C05497=1146.849,185.688,-61.263,-178.263,7.229,148.849
C05498=1146.844,185.937,-61.286,-178.260,7.230,148.849
C05499=1146.839,186.185,-61.308,-178.257,7.233,148.849
C05500=1146.835,186.434,-61.332,-178.255,7.235,148.849
C05501=1146.830,186.683,-61.355,-178.251,7.238,148.848
C05502=1146.825,186.932,-61.378,-178.249,7.240,148.848
C05503=1146.820,187.181,-61.402,-178.246,7.242,148.848
C05504=1146.816,187.430,-61.426,-178.244,7.244,148.848
C05505=1146.811,187.679,-61.449,-178.240,7.247,148.847
C05506=1146.807,187.928,-61.472,-178.238,7.249,148.847
C05507=1146.803,188.177,-61.495,-178.235,7.252,148.847
C05508=1146.798,188.426,-61.519,-178.232,7.253,148.846
C05509=1146.793,188.675,-61.542,-178.229,7.256,148.846
C05510=1146.789,188.923,-61.566,-178.227,7.258,148.846
C05511=1146.784,189.172,-61.590,-178.224,7.261,148.846
C05512=1146.780,189.421,-61.613,-178.221,7.263,148.845
C05513=1146.775,189.670,-61.636,-178.218,7.266,148.845
C05514=1146.770,189.919,-61.660,-178.216,7.267,148.845
C05515=1146.766,190.168,-61.684,-178.212,7.270,148.845
C05516=1146.761,190.417,-61.707,-178.210,7.272,148.845
C05517=1146.756,190.666,-61.730,-178.207,7.274,148.844
C05518=1146.752,190.914,-61.754,-178.205,7.277,148.844
C05519=1146.747,191.163,-61.778,-178.201,7.279,148.844
C05520=1146.743,191.412,-61.801,-178.199,7.281,148.844
C05521=1146.738,191.661,-61.825,-178.196,7.284,148.843
C05522=1146.733,191.910,-61.849,-178.194,7.286,148.843
C05523=1146.729,192.158,-61.873,-178.190,7.288,148.843
C05524=1146.724,192.407,-61.896,-178.188,7.291,148.843
C05525=1146.720,192.656,-61.919,-178.185,7.293,148.842
C05526=1146.715,192.904,-61.944,-178.182,7.296,148.842
C05527=1146.711,193.153,-61.967,-178.180,7.298,148.842
C05528=1146.706,193.402,-61.991,-178.177,7.301,148.842
C05529=1146.701,193.651,-62.014,-178.174,7.302,148.841
C05530=1146.697,193.899,-62.038,-178.171,7.305,148.841
C05531=1146.692,194.149,-62.062,-178.169,7.307,148.841
C05532=1146.688,194.398,-62.087,-178.165,7.310,148.841
C05533=1146.683,194.647,-62.110,-178.163,7.312,148.840
C05534=1146.679,194.895,-62.134,-178.160,7.314,148.840
C05535=1146.674,195.144,-62.158,-178.157,7.317,148.840
C05536=1146.670,195.393,-62.182,-178.154,7.319,148.840
C05537=1146.665,195.642,-62.205,-178.151,7.322,148.840
C05538=1146.661,195.890,-62.229,-178.149,7.324,148.839
C05539=1146.655,196.139,-62.253,-178.146,7.326,148.839
C05540=1146.651,196.388,-62.277,-178.143,7.328,148.839
C05541=1146.647,196.637,-62.302,-178.140,7.331,148.839
C05542=1146.642,196.886,-62.325,-178.138,7.333,148.838
C05543=1146.638,197.134,-62.349,-178.135,7.336,148.838
C05544=1146.632,197.384,-62.373,-178.132,7.338,148.838
C05545=1146.628,197.632,-62.397,-178.129,7.340,148.838
C05546=1146.624,197.881,-62.421,-178.127,7.343,148.838
C05547=1146.620,198.130,-62.445,-178.124,7.345,148.837
C05548=1146.615,198.379,-62.469,-178.121,7.348,148.837
C05549=1146.610,198.627,-62.494,-178.118,7.351,148.837
C05550=1146.606,198.876,-62.518,-178.116,7.353,148.837
C05551=1146.601,199.125,-62.541,-178.112,7.355,148.836
C05552=1146.596,199.374,-62.566,-178.110,7.357,148.836
C05553=1146.592,199.623,-62.590,-178.107,7.360,148.836
C05554=1146.588,199.871,-62.614,-178.104,7.363,148.836
C05555=1146.583,200.120,-62.638,-178.101,7.364,148.835
C05556=1146.578,200.369,-62.662,-178.099,7.367,148.835
C05557=1146.574,200.618,-62.687,-178.096,7.369,148.835
C05558=1146.570,200.866,-62.711,-178.093,7.372,148.835
C05559=1146.564,201.115,-62.735,-178.090,7.375,148.834
C05560=1146.560,201.364,-62.759,-178.088,7.377,148.834
C05561=1146.555,201.613,-62.783,-178.085,7.380,148.834
C05562=1146.551,201.862,-62.808,-178.082,7.381,148.834
C05563=1146.546,202.110,-62.832,-178.079,7.384,148.834
C05564=1146.542,202.359,-62.856,-178.076,7.387,148.833
C05565=1146.537,202.608,-62.881,-178.074,7.389,148.833
C05566=1146.533,202.857,-62.905,-178.071,7.391,148.833
C05567=1146.528,203.105,-62.930,-178.068,7.394,148.833
C05568=1146.524,203.354,-62.954,-178.066,7.397,148.833
C05569=1146.520,203.603,-62.978,-178.062,7.399,148.832
C05570=1146.515,203.852,-63.003,-178.060,7.401,148.832
C05571=1146.510,204.100,-63.027,-178.057,7.404,148.832
C05572=1146.506,204.350,-63.052,-178.054,7.407,148.832
C05573=1146.501,204.598,-63.076,-178.051,7.408,148.832
C05574=1146.496,204.847,-63.101,-178.049,7.411,148.831
C05575=1146.492,205.095,-63.125,-178.046,7.413,148.831
C05576=1146.488,205.344,-63.149,-178.043,7.416,148.831
C05577=1146.483,205.593,-63.174,-178.040,7.419,148.831
C05578=1146.478,205.841,-63.198,-178.038,7.421,148.831
C05579=1146.474,206.091,-63.223,-178.035,7.424,148.830
C05580=1146.469,206.339,-63.248,-178.032,7.426,148.830
C05581=1146.464,206.588,-63.272,-178.029,7.428,148.830
C05582=1146.460,206.837,-63.297,-178.027,7.431,148.830
C05583=1146.455,207.086,-63.321,-178.023,7.434,148.830
C05584=1146.451,207.334,-63.346,-178.021,7.436,148.829
C05585=1146.447,207.583,-63.371,-178.018,7.439,148.829
C05586=1146.442,207.832,-63.395,-178.015,7.441,148.829
C05587=1146.438,208.081,-63.420,-178.013,7.443,148.829
C05588=1146.433,208.330,-63.445,-178.010,7.446,148.829
C05589=1146.428,208.578,-63.469,-178.007,7.449,148.828
C05590=1146.424,208.827,-63.494,-178.004,7.451,148.828
C05591=1146.419,209.075,-63.519,-178.001,7.453,148.828
C05592=1146.415,209.346,-63.546,-177.998,7.456,148.828
C05593=1146.409,209.616,-63.573,-177.995,7.459,148.828
C05594=1146.405,209.887,-63.600,-177.992,7.462,148.827
C05595=1146.400,210.158,-63.627,-177.989,7.464,148.827
C05596=1146.395,210.407,-63.652,-177.986,7.467,148.827
C05597=1146.391,210.655,-63.676,-177.984,7.469,148.827
C05598=1146.387,210.904,-63.701,-177.981,7.472,148.827
C05599=1146.381,211.153,-63.726,-177.978,7.475,148.827
C05600=1146.377,211.401,-63.752,-177.976,7.477,148.826
C05601=1146.373,211.650,-63.776,-177.973,7.480,148.826
C05602=1146.368,211.899,-63.801,-177.970,7.483,148.826
C05603=1146.363,212.148,-63.826,-177.968,7.485,148.826
C05604=1146.359,212.396,-63.850,-177.964,7.487,148.826
C05605=1146.355,212.645,-63.876,-177.961,7.490,148.825
C05606=1146.350,212.894,-63.901,-177.959,7.492,148.825
C05607=1146.346,213.143,-63.925,-177.956,7.495,148.825
C05608=1146.341,213.391,-63.951,-177.953,7.498,148.825
C05609=1146.336,213.640,-63.976,-177.950,7.501,148.825
C05610=1146.332,213.888,-64.001,-177.948,7.502,148.824
C05611=1146.327,214.138,-64.026,-177.945,7.505,148.824
C05612=1146.323,214.386,-64.051,-177.942,7.508,148.824
C05613=1146.319,214.635,-64.076,-177.939,7.510,148.824
C05614=1146.314,214.883,-64.101,-177.937,7.513,148.824
C05615=1146.309,215.132,-64.127,-177.934,7.516,148.824
C05616=1146.304,215.381,-64.152,-177.931,7.519,148.824
C05617=1146.301,215.629,-64.177,-177.928,7.520,148.823
C05618=1146.296,215.878,-64.202,-177.926,7.523,148.823
C05619=1146.291,216.127,-64.227,-177.923,7.526,148.823
C05620=1146.287,216.376,-64.252,-177.920,7.528,148.823
C05621=1146.282,216.624,-64.278,-177.917,7.531,148.823
C05622=1146.278,216.873,-64.304,-177.914,7.534,148.823
C05623=1146.274,217.121,-64.328,-177.911,7.536,148.822
C05624=1146.269,217.370,-64.353,-177.909,7.539,148.822
C05625=1146.264,217.618,-64.379,-177.906,7.541,148.822
C05626=1146.260,217.868,-64.404,-177.903,7.544,148.822
C05627=1146.256,218.117,-64.430,-177.900,7.547,148.822
C05628=1146.251,218.365,-64.455,-177.898,7.549,148.822
C05629=1146.247,218.613,-64.481,-177.895,7.552,148.821
C05630=1146.242,218.863,-64.506,-177.892,7.554,148.821
C05631=1146.237,219.111,-64.531,-177.889,7.557,148.821
C05632=1146.233,219.360,-64.557,-177.887,7.560,148.821
C05633=1146.228,219.608,-64.582,-177.884,7.562,148.821
C05634=1146.224,219.857,-64.607,-177.881,7.565,148.820
C05635=1146.220,220.106,-64.632,-177.878,7.568,148.820
C05636=1146.215,220.354,-64.658,-177.876,7.570,148.820
C05637=1146.211,220.603,-64.684,-177.873,7.573,148.820
C05638=1146.207,220.851,-64.709,-177.870,7.576,148.820
C05639=1146.202,221.100,-64.735,-177.867,7.578,148.820
C05640=1146.198,221.348,-64.760,-177.865,7.581,148.820
C05641=1146.193,221.598,-64.786,-177.862,7.583,148.820
C05642=1146.188,221.846,-64.811,-177.859,7.586,148.819
C05643=1146.184,222.095,-64.837,-177.856,7.589,148.819
C05644=1146.179,222.344,-64.863,-177.854,7.591,148.819
C05645=1146.175,222.592,-64.888,-177.851,7.594,148.819
C05646=1146.170,222.841,-64.914,-177.848,7.597,148.819
C05647=1146.166,223.090,-64.940,-177.845,7.599,148.819
C05648=1146.161,223.338,-64.965,-177.842,7.602,148.818
C05649=1146.157,223.586,-64.991,-177.840,7.604,148.818
C05650=1146.153,223.835,-65.017,-177.837,7.607,148.818
C05651=1146.149,224.084,-65.043,-177.834,7.610,148.818
C05652=1146.144,224.332,-65.068,-177.831,7.613,148.818
C05653=1146.139,224.581,-65.094,-177.828,7.616,148.818
C05654=1146.135,224.830,-65.120,-177.826,7.618,148.818
C05655=1146.130,225.079,-65.146,-177.823,7.620,148.817
C05656=1146.126,225.327,-65.171,-177.820,7.623,148.817
C05657=1146.121,225.576,-65.197,-177.817,7.626,148.817
C05658=1146.117,225.824,-65.223,-177.814,7.629,148.817
C05659=1146.112,226.073,-65.250,-177.812,7.631,148.817
C05660=1146.108,226.321,-65.275,-177.809,7.634,148.817
C05661=1146.103,226.570,-65.301,-177.806,7.637,148.817
C05662=1146.099,226.819,-65.327,-177.803,7.640,148.816
C05663=1146.095,227.068,-65.352,-177.800,7.643,148.816
C05664=1146.089,227.316,-65.378,-177.798,7.645,148.816
C05665=1146.085,227.564,-65.405,-177.795,7.647,148.816
C05666=1146.081,227.813,-65.431,-177.792,7.650,148.816
C05667=1146.077,228.062,-65.456,-177.789,7.653,148.816
C05668=1146.072,228.311,-65.483,-177.787,7.656,148.816
C05669=1146.068,228.558,-65.509,-177.784,7.658,148.816
C05670=1146.063,228.807,-65.534,-177.782,7.661,148.816
C05671=1146.059,229.056,-65.560,-177.778,7.664,148.815
C05672=1146.054,229.305,-65.587,-177.776,7.667,148.815
C05673=1146.050,229.553,-65.613,-177.773,7.670,148.815
C05674=1146.046,229.802,-65.639,-177.770,7.672,148.815
C05675=1146.041,230.051,-65.665,-177.768,7.675,148.815
C05676=1146.036,230.299,-65.691,-177.765,7.677,148.815
C05677=1146.032,230.548,-65.717,-177.762,7.680,148.814
C05678=1146.027,230.797,-65.743,-177.759,7.683,148.814
C05679=1146.023,231.045,-65.770,-177.756,7.686,148.814
C05680=1146.019,231.294,-65.796,-177.753,7.689,148.814
C05681=1146.014,231.542,-65.823,-177.751,7.691,148.814
C05682=1146.010,231.791,-65.848,-177.748,7.694,148.814
C05683=1146.006,232.039,-65.875,-177.745,7.696,148.814
C05684=1146.001,232.288,-65.901,-177.742,7.699,148.814
C05685=1145.997,232.536,-65.927,-177.739,7.702,148.814
C05686=1145.992,232.785,-65.954,-177.737,7.705,148.813
C05687=1145.988,233.034,-65.979,-177.734,7.708,148.813
C05688=1145.983,233.282,-66.006,-177.732,7.710,148.813
C05689=1145.979,233.531,-66.032,-177.729,7.713,148.813
C05690=1145.975,233.779,-66.059,-177.726,7.716,148.813
C05691=1145.970,234.028,-66.086,-177.723,7.719,148.813
C05692=1145.966,234.276,-66.111,-177.720,7.722,148.813
C05693=1145.961,234.525,-66.139,-177.717,7.724,148.813
C05694=1145.957,234.774,-66.164,-177.714,7.727,148.813
C05695=1145.952,235.022,-66.191,-177.712,7.729,148.812
C05696=1145.948,235.294,-66.220,-177.709,7.733,148.812
C05697=1145.943,235.566,-66.249,-177.706,7.736,148.812
C05698=1145.938,235.837,-66.278,-177.703,7.739,148.812
C05699=1145.934,236.109,-66.307,-177.700,7.742,148.812
C05700=1145.929,236.358,-66.334,-177.697,7.745,148.812
C05701=1145.924,236.607,-66.361,-177.694,7.747,148.812
C05702=1145.920,236.855,-66.387,-177.692,7.750,148.812
C05703=1145.915,237.104,-66.413,-177.689,7.753,148.812
C05704=1145.911,237.352,-66.440,-177.686,7.756,148.811
C05705=1145.907,237.601,-66.467,-177.683,7.759,148.811
C05706=1145.903,237.849,-66.493,-177.680,7.762,148.811
C05707=1145.898,238.098,-66.520,-177.678,7.764,148.811
C05708=1145.893,238.347,-66.547,-177.675,7.767,148.811
C05709=1145.889,238.595,-66.573,-177.672,7.770,148.811
C05710=1145.885,238.843,-66.600,-177.669,7.773,148.811
C05711=1145.880,239.093,-66.627,-177.667,7.776,148.811
C05712=1145.876,239.341,-66.653,-177.664,7.778,148.811
C05713=1145.871,239.589,-66.680,-177.661,7.781,148.811
C05714=1145.866,239.838,-66.707,-177.658,7.784,148.810
C05715=1145.862,240.086,-66.734,-177.656,7.787,148.810
C05716=1145.858,240.334,-66.761,-177.653,7.790,148.810
C05717=1145.853,240.583,-66.788,-177.650,7.792,148.810
C05718=1145.849,240.831,-66.814,-177.647,7.795,148.810
C05719=1145.844,241.080,-66.841,-177.644,7.798,148.810
C05720=1145.840,241.329,-66.868,-177.642,7.801,148.810
C05721=1145.836,241.577,-66.894,-177.639,7.804,148.810
C05722=1145.832,241.826,-66.922,-177.636,7.807,148.810
C05723=1145.827,242.075,-66.949,-177.633,7.809,148.810
C05724=1145.822,242.323,-66.976,-177.631,7.812,148.809
C05725=1145.818,242.571,-67.002,-177.628,7.815,148.809
C05726=1145.814,242.820,-67.029,-177.625,7.818,148.809
C05727=1145.809,243.068,-67.056,-177.622,7.821,148.809
C05728=1145.804,243.317,-67.083,-177.619,7.824,148.809
C05729=1145.800,243.565,-67.110,-177.617,7.826,148.809
C05730=1145.797,243.813,-67.138,-177.614,7.829,148.809
C05731=1145.792,244.062,-67.165,-177.612,7.832,148.809
C05732=1145.787,244.310,-67.192,-177.609,7.835,148.809
C05733=1145.783,244.559,-67.219,-177.606,7.838,148.809
C05734=1145.778,244.807,-67.246,-177.603,7.841,148.809
C05735=1145.774,245.056,-67.273,-177.600,7.844,148.809
C05736=1145.770,245.305,-67.300,-177.598,7.847,148.809
C05737=1145.765,245.553,-67.327,-177.595,7.850,148.808
C05738=1145.761,245.801,-67.355,-177.592,7.853,148.808
C05739=1145.756,246.050,-67.382,-177.589,7.855,148.808
C05740=1145.752,246.298,-67.409,-177.586,7.858,148.808
C05741=1145.748,246.547,-67.437,-177.584,7.861,148.808
C05742=1145.743,246.796,-67.464,-177.581,7.864,148.808
C05743=1145.739,247.044,-67.491,-177.578,7.867,148.808
C05744=1145.735,247.292,-67.518,-177.575,7.870,148.808
C05745=1145.731,247.541,-67.545,-177.573,7.873,148.808
C05746=1145.726,247.790,-67.572,-177.570,7.875,148.808
C05747=1145.722,248.038,-67.600,-177.568,7.878,148.808
C05748=1145.717,248.286,-67.627,-177.565,7.881,148.808
C05749=1145.713,248.535,-67.655,-177.562,7.884,148.808
C05750=1145.709,248.783,-67.682,-177.559,7.887,148.807
C05751=1145.704,249.032,-67.709,-177.556,7.890,148.807
C05752=1145.699,249.280,-67.736,-177.554,7.893,148.807
C05753=1145.696,249.529,-67.765,-177.551,7.896,148.807
C05754=1145.691,249.777,-67.792,-177.548,7.898,148.807
C05755=1145.687,250.025,-67.819,-177.545,7.901,148.807
C05756=1145.682,250.274,-67.847,-177.542,7.904,148.807
C05757=1145.678,250.522,-67.875,-177.540,7.907,148.807
C05758=1145.674,250.771,-67.902,-177.537,7.910,148.807
C05759=1145.669,251.019,-67.929,-177.534,7.913,148.807
C05760=1145.665,251.268,-67.957,-177.531,7.916,148.807
C05761=1145.660,251.516,-67.985,-177.529,7.919,148.807
C05762=1145.655,251.764,-68.012,-177.526,7.922,148.807
C05763=1145.651,252.014,-68.040,-177.523,7.925,148.807
C05764=1145.647,252.261,-68.068,-177.520,7.928,148.806
C05765=1145.643,252.509,-68.095,-177.517,7.931,148.806
C05766=1145.639,252.758,-68.123,-177.515,7.934,148.806
C05767=1145.634,253.006,-68.151,-177.512,7.937,148.806
C05768=1145.630,253.255,-68.178,-177.509,7.939,148.806
C05769=1145.626,253.503,-68.206,-177.506,7.942,148.806
C05770=1145.620,253.752,-68.233,-177.503,7.945,148.806
C05771=1145.616,254.000,-68.261,-177.501,7.949,148.806
C05772=1145.612,254.249,-68.289,-177.498,7.951,148.806
C05773=1145.608,254.497,-68.316,-177.496,7.954,148.806
C05774=1145.604,254.746,-68.345,-177.493,7.957,148.806
C05775=1145.600,254.994,-68.372,-177.490,7.960,148.806
C05776=1145.594,255.242,-68.400,-177.487,7.963,148.806
C05777=1145.590,255.491,-68.428,-177.484,7.966,148.806
C05778=1145.586,255.739,-68.456,-177.482,7.969,148.806
C05779=1145.582,255.987,-68.484,-177.479,7.972,148.806
C05780=1145.577,256.236,-68.512,-177.476,7.975,148.806
C05781=1145.573,256.484,-68.539,-177.473,7.978,148.806
C05782=1145.569,256.733,-68.568,-177.470,7.981,148.805
C05783=1145.564,256.981,-68.595,-177.468,7.984,148.806
C05784=1145.560,257.230,-68.623,-177.465,7.987,148.806
C05785=1145.555,257.478,-68.651,-177.463,7.990,148.805
C05786=1145.552,257.727,-68.679,-177.460,7.993,148.805
C05787=1145.547,257.975,-68.708,-177.457,7.996,148.805
C05788=1145.543,258.223,-68.736,-177.454,7.999,148.805
C05789=1145.538,258.471,-68.764,-177.451,8.002,148.805
C05790=1145.534,258.720,-68.792,-177.449,8.005,148.805
C05791=1145.529,258.969,-68.819,-177.446,8.007,148.805
C05792=1145.526,259.217,-68.848,-177.444,8.011,148.805
C05793=1145.520,259.465,-68.876,-177.441,8.014,148.805
C05794=1145.517,259.714,-68.904,-177.438,8.017,148.805
C05795=1145.512,259.962,-68.932,-177.435,8.020,148.805
C05796=1145.508,260.211,-68.961,-177.432,8.022,148.805
C05797=1145.503,260.459,-68.988,-177.430,8.025,148.805
C05798=1145.500,260.707,-69.017,-177.427,8.028,148.805
C05799=1145.495,260.955,-69.045,-177.423,8.032,148.805
C05800=1145.490,261.229,-69.076,-177.421,8.035,148.805
C05801=1145.485,261.502,-69.107,-177.418,8.038,148.805
C05802=1145.481,261.776,-69.139,-177.415,8.042,148.805
C05803=1145.476,262.049,-69.169,-177.412,8.045,148.805
C05804=1145.471,262.297,-69.198,-177.409,8.048,148.805
C05805=1145.467,262.546,-69.226,-177.407,8.051,148.805
C05806=1145.463,262.795,-69.255,-177.404,8.054,148.805
C05807=1145.458,263.043,-69.282,-177.400,8.057,148.805
C05808=1145.454,263.291,-69.311,-177.398,8.061,148.805
C05809=1145.450,263.539,-69.340,-177.395,8.064,148.805
C05810=1145.445,263.788,-69.368,-177.393,8.067,148.805
C05811=1145.441,264.035,-69.396,-177.390,8.069,148.805
C05812=1145.437,264.284,-69.425,-177.387,8.072,148.805
C05813=1145.433,264.533,-69.453,-177.384,8.075,148.804
C05814=1145.428,264.781,-69.482,-177.382,8.079,148.805
C05815=1145.424,265.029,-69.511,-177.379,8.082,148.805
C05816=1145.419,265.277,-69.539,-177.376,8.084,148.805
C05817=1145.415,265.526,-69.567,-177.374,8.087,148.804
C05818=1145.411,265.774,-69.596,-177.371,8.090,148.804
C05819=1145.406,266.022,-69.625,-177.368,8.094,148.805
C05820=1145.402,266.271,-69.653,-177.366,8.097,148.804
C05821=1145.398,266.520,-69.681,-177.363,8.099,148.804
C05822=1145.393,266.767,-69.710,-177.359,8.103,148.804
C05823=1145.389,267.016,-69.739,-177.357,8.106,148.804
C05824=1145.385,267.264,-69.768,-177.354,8.109,148.805
C05825=1145.380,267.512,-69.796,-177.352,8.112,148.804
C05826=1145.376,267.761,-69.825,-177.349,8.115,148.804
C05827=1145.372,268.009,-69.854,-177.346,8.118,148.804
C05828=1145.367,268.257,-69.882,-177.344,8.121,148.804
C05829=1145.363,268.506,-69.911,-177.341,8.124,148.804
C05830=1145.359,268.754,-69.940,-177.338,8.127,148.804
C05831=1145.354,269.002,-69.968,-177.335,8.130,148.804
C05832=1145.351,269.250,-69.997,-177.333,8.133,148.804
C05833=1145.346,269.499,-70.026,-177.330,8.137,148.804
C05834=1145.341,269.747,-70.055,-177.327,8.140,148.804
C05835=1145.337,269.996,-70.084,-177.324,8.143,148.804
C05836=1145.334,270.244,-70.113,-177.321,8.146,148.804
C05837=1145.329,270.493,-70.141,-177.319,8.149,148.804
C05838=1145.324,270.740,-70.170,-177.316,8.152,148.804
C05839=1145.320,270.989,-70.199,-177.313,8.155,148.804
C05840=1145.316,271.237,-70.228,-177.311,8.158,148.804
C05841=1145.312,271.485,-70.258,-177.308,8.161,148.804
C05842=1145.307,271.733,-70.286,-177.305,8.164,148.804
C05843=1145.303,271.982,-70.315,-177.302,8.168,148.804
C05844=1145.299,272.230,-70.345,-177.300,8.171,148.805
C05845=1145.295,272.479,-70.373,-177.297,8.174,148.804
C05846=1145.290,272.726,-70.402,-177.294,8.177,148.804
C05847=1145.286,272.974,-70.432,-177.291,8.180,148.804
C05848=1145.281,273.223,-70.460,-177.289,8.183,148.805
C05849=1145.277,273.472,-70.490,-177.286,8.186,148.804
C05850=1145.273,273.720,-70.519,-177.284,8.189,148.804
C05851=1145.268,273.968,-70.548,-177.281,8.193,148.805
C05852=1145.265,274.216,-70.576,-177.278,8.196,148.805
C05853=1145.260,274.464,-70.606,-177.275,8.199,148.805
C05854=1145.256,274.712,-70.635,-177.272,8.202,148.804
C05855=1145.252,274.961,-70.664,-177.270,8.205,148.805
C05856=1145.248,275.210,-70.693,-177.267,8.208,148.805
C05857=1145.243,275.457,-70.723,-177.264,8.211,148.805
C05858=1145.239,275.705,-70.752,-177.262,8.215,148.805
C05859=1145.234,275.954,-70.781,-177.259,8.218,148.805
C05860=1145.230,276.202,-70.811,-177.256,8.221,148.805
C05861=1145.226,276.451,-70.840,-177.254,8.224,148.805
C05862=1145.222,276.699,-70.869,-177.251,8.227,148.805
C05863=1145.217,276.947,-70.899,-177.248,8.230,148.805
C05864=1145.213,277.196,-70.928,-177.246,8.234,148.805
C05865=1145.208,277.443,-70.957,-177.243,8.237,148.805
C05866=1145.204,277.692,-70.987,-177.240,8.240,148.805
C05867=1145.200,277.940,-71.016,-177.237,8.244,148.805
C05868=1145.196,278.188,-71.045,-177.234,8.246,148.805
C05869=1145.192,278.436,-71.075,-177.232,8.249,148.805
C05870=1145.187,278.685,-71.104,-177.229,8.253,148.805
C05871=1145.183,278.933,-71.134,-177.227,8.256,148.805
C05872=1145.179,279.181,-71.163,-177.223,8.259,148.805
C05873=1145.175,279.429,-71.193,-177.221,8.263,148.805
C05874=1145.171,279.678,-71.222,-177.218,8.266,148.805
C05875=1145.167,279.926,-71.252,-177.215,8.268,148.805
C05876=1145.162,280.174,-71.281,-177.213,8.272,148.805
C05877=1145.158,280.422,-71.311,-177.210,8.275,148.805
C05878=1145.154,280.671,-71.340,-177.207,8.279,148.805
C05879=1145.149,280.919,-71.370,-177.204,8.282,148.805
C05880=1145.145,281.166,-71.400,-177.202,8.285,148.805
C05881=1145.140,281.415,-71.429,-177.199,8.288,148.805
C05882=1145.136,281.663,-71.459,-177.197,8.291,148.805
C05883=1145.132,281.911,-71.488,-177.194,8.294,148.805
C05884=1145.128,282.159,-71.518,-177.191,8.298,148.805
C05885=1145.124,282.408,-71.547,-177.188,8.301,148.805
C05886=1145.119,282.656,-71.578,-177.186,8.304,148.806
C05887=1145.115,282.904,-71.607,-177.183,8.307,148.806
C05888=1145.111,283.152,-71.637,-177.181,8.310,148.806
C05889=1145.107,283.400,-71.666,-177.178,8.313,148.806
C05890=1145.102,283.648,-71.697,-177.175,8.317,148.806
C05891=1145.098,283.897,-71.726,-177.172,8.320,148.806
C05892=1145.094,284.145,-71.756,-177.169,8.323,148.806
C05893=1145.090,284.393,-71.786,-177.167,8.326,148.806
C05894=1145.085,284.642,-71.817,-177.164,8.329,148.806
C05895=1145.081,284.890,-71.846,-177.161,8.333,148.806
C05896=1145.077,285.138,-71.876,-177.159,8.336,148.806
C05897=1145.073,285.386,-71.906,-177.156,8.339,148.806
C05898=1145.068,285.635,-71.936,-177.154,8.343,148.806
C05899=1145.064,285.882,-71.966,-177.151,8.345,148.806
C05900=1145.060,286.130,-71.995,-177.148,8.350,148.806
C05901=1145.056,286.378,-72.026,-177.145,8.352,148.806
C05902=1145.051,286.627,-72.055,-177.143,8.356,148.806
C05903=1145.048,286.874,-72.086,-177.140,8.359,148.806
C05904=1145.042,287.151,-72.119,-177.137,8.363,148.807
C05905=1145.038,287.426,-72.153,-177.134,8.367,148.807
C05906=1145.033,287.702,-72.185,-177.131,8.369,148.807
C05907=1145.029,287.976,-72.219,-177.128,8.374,148.807
C05908=1145.024,288.225,-72.249,-177.125,8.376,148.807
C05909=1145.020,288.473,-72.279,-177.123,8.380,148.807
C05910=1145.015,288.721,-72.310,-177.120,8.383,148.807
C05911=1145.012,288.970,-72.340,-177.117,8.387,148.807
C05912=1145.008,289.217,-72.370,-177.114,8.390,148.807
C05913=1145.003,289.466,-72.400,-177.112,8.393,148.807
C05914=1144.999,289.713,-72.430,-177.109,8.397,148.807
C05915=1144.995,289.961,-72.461,-177.106,8.400,148.807
C05916=1144.990,290.210,-72.490,-177.104,8.403,148.807
C05917=1144.986,290.458,-72.521,-177.101,8.406,148.807
C05918=1144.982,290.706,-72.552,-177.098,8.409,148.807
C05919=1144.978,290.955,-72.582,-177.096,8.413,148.808
C05920=1144.974,291.202,-72.612,-177.093,8.416,148.808
C05921=1144.969,291.450,-72.642,-177.090,8.419,148.808
C05922=1144.965,291.698,-72.672,-177.088,8.422,148.808
C05923=1144.961,291.947,-72.703,-177.085,8.426,148.808
C05924=1144.957,292.195,-72.733,-177.082,8.429,148.808
C05925=1144.952,292.443,-72.764,-177.080,8.433,148.808
C05926=1144.949,292.690,-72.794,-177.077,8.436,148.808
C05927=1144.944,292.940,-72.825,-177.074,8.440,148.808
C05928=1144.940,293.187,-72.855,-177.072,8.443,148.808
C05929=1144.936,293.435,-72.886,-177.069,8.446,148.808
C05930=1144.931,293.683,-72.916,-177.067,8.449,148.809
C05931=1144.928,293.931,-72.947,-177.063,8.453,148.809
C05932=1144.923,294.179,-72.978,-177.061,8.456,148.809
C05933=1144.919,294.428,-73.007,-177.058,8.459,148.809
C05934=1144.914,294.676,-73.038,-177.056,8.462,148.809
C05935=1144.910,294.924,-73.069,-177.053,8.466,148.809
C05936=1144.907,295.172,-73.099,-177.050,8.469,148.809
C05937=1144.902,295.420,-73.130,-177.048,8.473,148.809
C05938=1144.898,295.669,-73.161,-177.045,8.476,148.809
C05939=1144.894,295.916,-73.191,-177.042,8.480,148.809
C05940=1144.889,296.164,-73.222,-177.039,8.483,148.809
C05941=1144.886,296.412,-73.252,-177.037,8.486,148.810
C05942=1144.882,296.661,-73.283,-177.035,8.489,148.810
C05943=1144.877,296.908,-73.314,-177.031,8.493,148.810
C05944=1144.872,297.156,-73.345,-177.029,8.496,148.810
C05945=1144.869,297.405,-73.375,-177.026,8.499,148.810
C05946=1144.864,297.653,-73.406,-177.023,8.503,148.810
C05947=1144.860,297.901,-73.437,-177.021,8.506,148.810
C05948=1144.856,298.149,-73.468,-177.018,8.509,148.810
C05949=1144.852,298.396,-73.499,-177.016,8.513,148.810
C05950=1144.848,298.644,-73.530,-177.013,8.517,148.811
C05951=1144.844,298.893,-73.561,-177.010,8.520,148.811
C05952=1144.839,299.141,-73.591,-177.008,8.523,148.811
C05953=1144.836,299.389,-73.622,-177.004,8.527,148.811
C05954=1144.831,299.637,-73.653,-177.002,8.530,148.811
C05955=1144.827,299.885,-73.684,-177.000,8.533,148.811
C05956=1144.823,300.133,-73.715,-176.997,8.536,148.811
C05957=1144.818,300.381,-73.746,-176.994,8.540,148.811
C05958=1144.814,300.630,-73.777,-176.992,8.543,148.811
C05959=1144.810,300.878,-73.807,-176.989,8.546,148.811
C05960=1144.806,301.125,-73.839,-176.986,8.550,148.812
C05961=1144.802,301.374,-73.870,-176.984,8.554,148.812
C05962=1144.797,301.621,-73.901,-176.981,8.557,148.812
C05963=1144.794,301.870,-73.933,-176.978,8.561,148.812
C05964=1144.789,302.117,-73.963,-176.976,8.564,148.812
C05965=1144.784,302.365,-73.994,-176.973,8.567,148.812
C05966=1144.781,302.613,-74.026,-176.971,8.570,148.812
C05967=1144.776,302.861,-74.057,-176.968,8.574,148.812
C05968=1144.772,303.110,-74.088,-176.965,8.577,148.812
C05969=1144.768,303.357,-74.119,-176.963,8.580,148.813
C05970=1144.764,303.606,-74.150,-176.960,8.585,148.813
C05971=1144.760,303.853,-74.181,-176.957,8.588,148.813
C05972=1144.756,304.102,-74.213,-176.955,8.591,148.813
C05973=1144.752,304.350,-74.243,-176.952,8.595,148.813
C05974=1144.748,304.598,-74.275,-176.949,8.598,148.813
C05975=1144.743,304.846,-74.306,-176.947,8.601,148.813
C05976=1144.739,305.093,-74.337,-176.944,8.605,148.814
C05977=1144.735,305.342,-74.369,-176.941,8.608,148.814
C05978=1144.731,305.589,-74.400,-176.939,8.612,148.814
C05979=1144.726,305.838,-74.432,-176.936,8.615,148.814
C05980=1144.722,306.086,-74.464,-176.933,8.619,148.814
C05981=1144.718,306.333,-74.495,-176.931,8.622,148.814
C05982=1144.714,306.582,-74.526,-176.928,8.626,148.815
C05983=1144.710,306.829,-74.558,-176.925,8.629,148.815
C05984=1144.706,307.078,-74.589,-176.923,8.632,148.815
C05985=1144.701,307.325,-74.620,-176.920,8.636,148.815
C05986=1144.698,307.573,-74.652,-176.918,8.640,148.815
C05987=1144.693,307.821,-74.683,-176.915,8.643,148.815
C05988=1144.689,308.069,-74.715,-176.912,8.647,148.815
C05989=1144.685,308.317,-74.746,-176.910,8.650,148.815
C05990=1144.680,308.566,-74.778,-176.907,8.653,148.816
C05991=1144.676,308.814,-74.810,-176.904,8.657,148.816
C05992=1144.672,309.061,-74.841,-176.902,8.660,148.816
C05993=1144.668,309.309,-74.873,-176.899,8.663,148.816
C05994=1144.664,309.557,-74.904,-176.896,8.667,148.816
C05995=1144.660,309.805,-74.936,-176.894,8.671,148.816
C05996=1144.656,310.053,-74.968,-176.891,8.675,148.816
C05997=1144.651,310.301,-75.000,-176.888,8.678,148.817
C05998=1144.647,310.549,-75.031,-176.886,8.681,148.817
C05999=1144.643,310.797,-75.062,-176.883,8.685,148.817
C06000=1144.639,311.045,-75.094,-176.881,8.688,148.817
C06001=1144.635,311.293,-75.127,-176.878,8.692,148.817
C06002=1144.631,311.541,-75.158,-176.875,8.695,148.817
C06003=1144.627,311.789,-75.190,-176.873,8.699,148.818
C06004=1144.623,312.037,-75.222,-176.870,8.702,148.818
C06005=1144.618,312.284,-75.254,-176.867,8.706,148.818
C06006=1144.614,312.533,-75.285,-176.865,8.709,148.818
C06007=1144.610,312.781,-75.317,-176.862,8.713,148.818
C06008=1144.606,313.059,-75.352,-176.859,8.717,148.818
C06009=1144.601,313.336,-75.389,-176.857,8.720,148.819
C06010=1144.597,313.614,-75.424,-176.854,8.724,148.819
C06011=1144.592,313.892,-75.460,-176.851,8.729,148.819
C06012=1144.587,314.139,-75.492,-176.848,8.733,148.819
C06013=1144.584,314.387,-75.524,-176.845,8.736,148.819
C06014=1144.579,314.635,-75.556,-176.843,8.739,148.820
C06015=1144.575,314.883,-75.588,-176.840,8.743,148.820
C06016=1144.571,315.131,-75.619,-176.837,8.746,148.820
C06017=1144.567,315.379,-75.652,-176.835,8.750,148.820
C06018=1144.563,315.627,-75.684,-176.832,8.754,148.820
C06019=1144.559,315.875,-75.715,-176.830,8.757,148.820
C06020=1144.555,316.122,-75.748,-176.827,8.761,148.821
C06021=1144.551,316.370,-75.780,-176.825,8.764,148.821
C06022=1144.546,316.619,-75.813,-176.822,8.768,148.821
C06023=1144.542,316.866,-75.844,-176.819,8.771,148.821
C06024=1144.538,317.114,-75.877,-176.817,8.774,148.821
C06025=1144.534,317.362,-75.908,-176.814,8.779,148.821
C06026=1144.531,317.610,-75.941,-176.811,8.782,148.822
C06027=1144.526,317.858,-75.973,-176.808,8.786,148.822
C06028=1144.522,318.105,-76.005,-176.806,8.789,148.822
C06029=1144.517,318.354,-76.037,-176.804,8.792,148.822
C06030=1144.514,318.601,-76.070,-176.801,8.796,148.822
C06031=1144.510,318.850,-76.102,-176.799,8.800,148.823
C06032=1144.506,319.098,-76.134,-176.796,8.804,148.823
C06033=1144.501,319.345,-76.167,-176.793,8.807,148.823
C06034=1144.497,319.593,-76.199,-176.790,8.811,148.823
C06035=1144.493,319.841,-76.231,-176.788,8.814,148.824
C06036=1144.490,320.088,-76.264,-176.786,8.818,148.824
C06037=1144.485,320.337,-76.296,-176.783,8.822,148.824
C06038=1144.481,320.585,-76.328,-176.780,8.825,148.824
C06039=1144.477,320.832,-76.361,-176.778,8.829,148.824
C06040=1144.472,321.080,-76.393,-176.775,8.832,148.825
C06041=1144.469,321.328,-76.426,-176.772,8.836,148.825
C06042=1144.464,321.576,-76.458,-176.770,8.840,148.825
C06043=1144.461,321.823,-76.491,-176.768,8.843,148.825
C06044=1144.456,322.072,-76.523,-176.765,8.847,148.825
C06045=1144.452,322.320,-76.557,-176.762,8.850,148.826
C06046=1144.449,322.568,-76.588,-176.759,8.854,148.826
C06047=1144.445,322.815,-76.622,-176.757,8.858,148.826
C06048=1144.439,323.063,-76.654,-176.754,8.862,148.826
C06049=1144.436,323.310,-76.686,-176.752,8.865,148.826
C06050=1144.432,323.559,-76.719,-176.749,8.869,148.827
C06051=1144.428,323.806,-76.751,-176.747,8.872,148.827
C06052=1144.424,324.054,-76.784,-176.744,8.876,148.827
C06053=1144.420,324.302,-76.817,-176.741,8.880,148.827
C06054=1144.416,324.550,-76.850,-176.739,8.883,148.827
C06055=1144.412,324.797,-76.882,-176.736,8.887,148.828
C06056=1144.408,325.046,-76.915,-176.734,8.890,148.828
C06057=1144.404,325.293,-76.948,-176.731,8.894,148.828
C06058=1144.400,325.541,-76.981,-176.729,8.898,148.828
C06059=1144.396,325.789,-77.013,-176.726,8.902,148.829
C06060=1144.392,326.037,-77.046,-176.723,8.905,148.829
C06061=1144.387,326.285,-77.079,-176.720,8.909,148.829
C06062=1144.383,326.533,-77.112,-176.718,8.912,148.829
C06063=1144.380,326.780,-77.144,-176.715,8.916,148.829
C06064=1144.375,327.028,-77.178,-176.713,8.920,148.830
C06065=1144.371,327.276,-77.211,-176.710,8.924,148.830
C06066=1144.367,327.524,-77.244,-176.708,8.927,148.830
C06067=1144.363,327.772,-77.276,-176.705,8.931,148.830
C06068=1144.359,328.019,-77.309,-176.703,8.935,148.831
C06069=1144.355,328.267,-77.342,-176.700,8.938,148.831
C06070=1144.351,328.515,-77.375,-176.697,8.942,148.831
C06071=1144.347,328.763,-77.408,-176.695,8.945,148.831
C06072=1144.343,329.010,-77.441,-176.692,8.949,148.831
C06073=1144.339,329.258,-77.475,-176.690,8.953,148.832
C06074=1144.334,329.506,-77.507,-176.687,8.957,148.832
C06075=1144.330,329.754,-77.540,-176.685,8.960,148.832
C06076=1144.326,330.002,-77.573,-176.682,8.964,148.832
C06077=1144.322,330.249,-77.606,-176.680,8.968,148.833
C06078=1144.318,330.497,-77.639,-176.677,8.972,148.833
C06079=1144.314,330.745,-77.672,-176.675,8.975,148.833
C06080=1144.310,330.992,-77.705,-176.672,8.979,148.833
C06081=1144.306,331.240,-77.739,-176.669,8.982,148.834
C06082=1144.302,331.488,-77.772,-176.666,8.986,148.834
C06083=1144.298,331.736,-77.805,-176.664,8.990,148.834
C06084=1144.294,331.984,-77.838,-176.662,8.994,148.834
C06085=1144.290,332.231,-77.872,-176.659,8.997,148.835
C06086=1144.286,332.479,-77.905,-176.656,9.001,148.835
C06087=1144.282,332.727,-77.939,-176.654,9.005,148.835
C06088=1144.278,332.974,-77.972,-176.651,9.009,148.835
C06089=1144.274,333.222,-78.005,-176.648,9.013,148.836
C06090=1144.270,333.470,-78.038,-176.646,9.016,148.836
C06091=1144.265,333.718,-78.071,-176.643,9.021,148.836
C06092=1144.262,333.965,-78.105,-176.641,9.024,148.836
C06093=1144.258,334.213,-78.139,-176.638,9.028,148.837
C06094=1144.254,334.461,-78.172,-176.636,9.031,148.837
C06095=1144.249,334.709,-78.206,-176.633,9.035,148.837
C06096=1144.245,334.957,-78.239,-176.631,9.039,148.837
C06097=1144.241,335.204,-78.273,-176.628,9.043,148.838
C06098=1144.237,335.451,-78.306,-176.626,9.046,148.838
C06099=1144.233,335.700,-78.339,-176.623,9.050,148.838
C06100=1144.230,335.947,-78.373,-176.620,9.053,148.838
C06101=1144.225,336.195,-78.406,-176.618,9.058,148.839
C06102=1144.221,336.442,-78.439,-176.616,9.061,148.839
C06103=1144.217,336.690,-78.473,-176.613,9.065,148.839
C06104=1144.213,336.938,-78.507,-176.610,9.068,148.839
C06105=1144.209,337.186,-78.541,-176.608,9.073,148.840
C06106=1144.205,337.433,-78.574,-176.605,9.077,148.840
C06107=1144.201,337.681,-78.608,-176.603,9.080,148.840
C06108=1144.198,337.929,-78.642,-176.600,9.084,148.841
C06109=1144.193,338.177,-78.676,-176.598,9.088,148.841
C06110=1144.189,338.424,-78.709,-176.595,9.092,148.841
C06111=1144.185,338.672,-78.743,-176.592,9.095,148.841
C06112=1144.180,338.952,-78.781,-176.590,9.099,148.842
C06113=1144.176,339.232,-78.819,-176.587,9.104,148.842
C06114=1144.172,339.513,-78.857,-176.584,9.109,148.842
C06115=1144.167,339.794,-78.896,-176.581,9.113,148.843
C06116=1144.163,340.041,-78.929,-176.578,9.117,148.843
C06117=1144.159,340.288,-78.963,-176.576,9.120,148.843
C06118=1144.155,340.537,-78.997,-176.573,9.124,148.844
C06119=1144.151,340.784,-79.031,-176.571,9.128,148.844
C06120=1144.147,341.031,-79.065,-176.568,9.132,148.844
C06121=1144.143,341.280,-79.099,-176.566,9.135,148.844
C06122=1144.139,341.527,-79.133,-176.563,9.139,148.845
C06123=1144.135,341.775,-79.166,-176.560,9.144,148.845
C06124=1144.130,342.022,-79.200,-176.558,9.147,148.845
C06125=1144.127,342.270,-79.235,-176.555,9.151,148.846
C06126=1144.123,342.518,-79.268,-176.553,9.155,148.846
C06127=1144.118,342.765,-79.302,-176.550,9.159,148.846
C06128=1144.115,343.013,-79.337,-176.548,9.162,148.846
C06129=1144.110,343.261,-79.371,-176.545,9.166,148.847
C06130=1144.106,343.508,-79.404,-176.543,9.171,148.847
C06131=1144.102,343.756,-79.439,-176.540,9.174,148.847
C06132=1144.098,344.004,-79.473,-176.538,9.178,148.848
C06133=1144.095,344.251,-79.507,-176.535,9.181,148.848
C06134=1144.091,344.499,-79.542,-176.532,9.186,148.848
C06135=1144.086,344.747,-79.575,-176.530,9.190,148.849
C06136=1144.083,344.995,-79.610,-176.528,9.193,148.849
C06137=1144.079,345.242,-79.643,-176.525,9.197,148.849
C06138=1144.074,345.489,-79.678,-176.523,9.201,148.849
C06139=1144.071,345.737,-79.712,-176.520,9.205,148.850
C06140=1144.066,345.984,-79.747,-176.517,9.209,148.850
C06141=1144.063,346.232,-79.781,-176.515,9.213,148.850
C06142=1144.059,346.480,-79.815,-176.512,9.217,148.851
C06143=1144.055,346.728,-79.849,-176.510,9.220,148.851
C06144=1144.050,346.976,-79.883,-176.507,9.224,148.851
C06145=1144.047,347.223,-79.917,-176.504,9.228,148.852
C06146=1144.043,347.471,-79.952,-176.502,9.232,148.852
C06147=1144.038,347.718,-79.986,-176.500,9.236,148.852
C06148=1144.035,347.966,-80.021,-176.497,9.240,148.853
C06149=1144.030,348.213,-80.055,-176.495,9.244,148.853
C06150=1144.027,348.461,-80.089,-176.492,9.248,148.853
C06151=1144.023,348.708,-80.125,-176.490,9.251,148.854
C06152=1144.019,348.956,-80.159,-176.487,9.255,148.854
C06153=1144.015,349.203,-80.193,-176.484,9.260,148.854
C06154=1144.011,349.451,-80.228,-176.482,9.263,148.854
C06155=1144.007,349.698,-80.262,-176.480,9.267,148.855
C06156=1144.003,349.947,-80.297,-176.477,9.272,148.855
C06157=1143.999,350.194,-80.331,-176.474,9.275,148.855
C06158=1143.995,350.442,-80.366,-176.472,9.279,148.856
C06159=1143.991,350.689,-80.401,-176.470,9.282,148.856
C06160=1143.987,350.937,-80.436,-176.467,9.287,148.856
C06161=1143.983,351.184,-80.469,-176.464,9.291,148.857
C06162=1143.979,351.432,-80.504,-176.462,9.295,148.857
C06163=1143.975,351.679,-80.539,-176.459,9.299,148.857
C06164=1143.971,351.927,-80.574,-176.457,9.303,148.858
C06165=1143.967,352.174,-80.608,-176.454,9.306,148.858
C06166=1143.963,352.422,-80.643,-176.452,9.310,148.858
C06167=1143.959,352.669,-80.678,-176.449,9.315,148.859
C06168=1143.955,352.917,-80.713,-176.447,9.318,148.859
C06169=1143.952,353.165,-80.747,-176.444,9.322,148.859
C06170=1143.948,353.412,-80.782,-176.441,9.326,148.860
C06171=1143.944,353.660,-80.817,-176.439,9.330,148.860
C06172=1143.939,353.907,-80.852,-176.436,9.334,148.860
C06173=1143.936,354.154,-80.887,-176.434,9.339,148.861
C06174=1143.932,354.402,-80.921,-176.432,9.342,148.861
C06175=1143.928,354.649,-80.957,-176.429,9.346,148.861
C06176=1143.924,354.897,-80.992,-176.426,9.350,148.862
C06177=1143.919,355.145,-81.026,-176.424,9.354,148.862
C06178=1143.916,355.392,-81.062,-176.421,9.358,148.862
C06179=1143.912,355.640,-81.096,-176.419,9.362,148.863
C06180=1143.908,355.887,-81.131,-176.417,9.366,148.863
C06181=1143.904,356.135,-81.166,-176.414,9.370,148.863
C06182=1143.901,356.383,-81.201,-176.411,9.374,148.864
C06183=1143.896,356.630,-81.236,-176.409,9.378,148.864
C06184=1143.892,356.877,-81.271,-176.406,9.382,148.864
C06185=1143.888,357.124,-81.307,-176.404,9.386,148.865
C06186=1143.884,357.372,-81.341,-176.401,9.389,148.865
C06187=1143.880,357.620,-81.377,-176.399,9.394,148.866
C06188=1143.877,357.868,-81.411,-176.396,9.398,148.866
C06189=1143.873,358.115,-81.446,-176.394,9.401,148.866
C06190=1143.869,358.362,-81.482,-176.392,9.406,148.867
C06191=1143.865,358.610,-81.517,-176.389,9.410,148.867
C06192=1143.861,358.857,-81.552,-176.386,9.414,148.867
C06193=1143.857,359.104,-81.587,-176.384,9.418,148.868
C06194=1143.853,359.353,-81.622,-176.381,9.422,148.868
C06195=1143.849,359.599,-81.657,-176.378,9.426,148.868
C06196=1143.845,359.847,-81.693,-176.376,9.430,148.869
C06197=1143.842,360.094,-81.729,-176.374,9.434,148.869
C06198=1143.838,360.342,-81.763,-176.371,9.438,148.869
C06199=1143.834,360.589,-81.799,-176.368,9.442,148.870
C06200=1143.830,360.837,-81.834,-176.366,9.446,148.870
C06201=1143.826,361.084,-81.870,-176.363,9.450,148.870
C06202=1143.823,361.332,-81.905,-176.361,9.454,148.871
C06203=1143.819,361.579,-81.941,-176.358,9.459,148.871
C06204=1143.814,361.827,-81.976,-176.355,9.463,148.872
C06205=1143.810,362.075,-82.011,-176.353,9.467,148.872
C06206=1143.806,362.322,-82.047,-176.351,9.470,148.872
C06207=1143.803,362.570,-82.082,-176.348,9.475,148.873
C06208=1143.798,362.816,-82.118,-176.345,9.479,148.873
C06209=1143.795,363.064,-82.153,-176.343,9.483,148.873
C06210=1143.791,363.311,-82.189,-176.340,9.487,148.874
C06211=1143.787,363.559,-82.224,-176.338,9.491,148.874
C06212=1143.784,363.806,-82.260,-176.335,9.495,148.874
C06213=1143.779,364.054,-82.296,-176.332,9.499,148.875
C06214=1143.775,364.301,-82.331,-176.329,9.503,148.875
C06215=1143.771,364.548,-82.367,-176.327,9.508,148.876
C06216=1143.767,364.832,-82.407,-176.323,9.513,148.876
C06217=1143.763,365.116,-82.449,-176.321,9.517,148.876
C06218=1143.759,365.399,-82.489,-176.318,9.522,148.877
C06219=1143.754,365.683,-82.530,-176.315,9.526,148.877
C06220=1143.750,365.930,-82.566,-176.312,9.531,148.878
C06221=1143.746,366.178,-82.602,-176.310,9.535,148.878
C06222=1143.743,366.425,-82.637,-176.307,9.539,148.878
C06223=1143.738,366.672,-82.673,-176.305,9.544,148.879
C06224=1143.734,366.919,-82.709,-176.302,9.548,148.879
C06225=1143.731,367.167,-82.745,-176.299,9.552,148.880
C06226=1143.727,367.414,-82.781,-176.296,9.556,148.880
C06227=1143.723,367.662,-82.817,-176.294,9.560,148.880
C06228=1143.719,367.910,-82.852,-176.291,9.565,148.881
C06229=1143.715,368.157,-82.889,-176.288,9.569,148.881
C06230=1143.711,368.404,-82.925,-176.286,9.572,148.881
C06231=1143.707,368.652,-82.960,-176.283,9.577,148.882
C06232=1143.704,368.899,-82.996,-176.281,9.581,148.882
C06233=1143.700,369.147,-83.033,-176.278,9.585,148.883
C06234=1143.696,369.394,-83.068,-176.275,9.589,148.883
C06235=1143.693,369.641,-83.104,-176.273,9.594,148.883
C06236=1143.688,369.888,-83.140,-176.270,9.598,148.884
C06237=1143.684,370.136,-83.176,-176.267,9.602,148.884
C06238=1143.680,370.383,-83.213,-176.265,9.607,148.885
C06239=1143.676,370.630,-83.248,-176.262,9.611,148.885
C06240=1143.673,370.877,-83.284,-176.260,9.615,148.885
C06241=1143.668,371.125,-83.321,-176.257,9.619,148.886
C06242=1143.665,371.372,-83.357,-176.255,9.623,148.886
C06243=1143.661,371.620,-83.393,-176.253,9.627,148.887
C06244=1143.657,371.867,-83.429,-176.250,9.632,148.887
C06245=1143.653,372.114,-83.465,-176.247,9.636,148.887
C06246=1143.650,372.361,-83.502,-176.245,9.640,148.888
C06247=1143.645,372.609,-83.538,-176.242,9.645,148.888
C06248=1143.642,372.856,-83.574,-176.240,9.649,148.889
C06249=1143.638,373.104,-83.611,-176.238,9.653,148.889
C06250=1143.635,373.351,-83.647,-176.235,9.657,148.889
C06251=1143.630,373.599,-83.683,-176.232,9.661,148.890
C06252=1143.627,373.846,-83.719,-176.230,9.665,148.890
C06253=1143.623,374.093,-83.756,-176.227,9.670,148.891
C06254=1143.619,374.341,-83.792,-176.225,9.673,148.891
C06255=1143.615,374.588,-83.828,-176.223,9.678,148.892
C06256=1143.611,374.835,-83.865,-176.220,9.682,148.892
C06257=1143.607,375.083,-83.901,-176.218,9.687,148.893
C06258=1143.603,375.330,-83.938,-176.216,9.690,148.893
C06259=1143.600,375.577,-83.974,-176.213,9.695,148.894
C06260=1143.596,375.824,-84.011,-176.211,9.699,148.894
C06261=1143.591,376.072,-84.047,-176.209,9.703,148.895
C06262=1143.589,376.319,-84.084,-176.207,9.707,148.895
C06263=1143.585,376.566,-84.120,-176.205,9.711,148.896
C06264=1143.580,376.814,-84.157,-176.203,9.715,148.896
C06265=1143.577,377.061,-84.194,-176.201,9.719,148.897
C06266=1143.573,377.308,-84.230,-176.199,9.723,148.897
C06267=1143.569,377.556,-84.267,-176.197,9.727,148.897
C06268=1143.565,377.802,-84.303,-176.194,9.732,148.898
C06269=1143.561,378.050,-84.340,-176.193,9.735,148.899
C06270=1143.558,378.297,-84.377,-176.191,9.739,148.899
C06271=1143.554,378.544,-84.413,-176.189,9.744,148.900
C06272=1143.550,378.792,-84.450,-176.187,9.747,148.900
C06273=1143.546,379.039,-84.487,-176.185,9.751,148.901
C06274=1143.542,379.287,-84.523,-176.183,9.756,148.901
C06275=1143.538,379.533,-84.559,-176.182,9.760,148.902
C06276=1143.534,379.781,-84.596,-176.180,9.763,148.902
C06277=1143.531,380.029,-84.633,-176.178,9.767,148.903
C06278=1143.527,380.276,-84.670,-176.177,9.771,148.904
C06279=1143.523,380.523,-84.707,-176.175,9.775,148.904
C06280=1143.519,380.770,-84.743,-176.173,9.778,148.905
C06281=1143.515,381.017,-84.780,-176.172,9.782,148.905
C06282=1143.512,381.265,-84.817,-176.170,9.786,148.906
C06283=1143.508,381.512,-84.854,-176.169,9.789,148.906
C06284=1143.504,381.759,-84.891,-176.168,9.793,148.907
C06285=1143.500,382.005,-84.928,-176.166,9.797,148.908
C06286=1143.496,382.253,-84.965,-176.166,9.800,148.908
C06287=1143.493,382.501,-85.002,-176.164,9.804,148.909
C06288=1143.489,382.747,-85.039,-176.163,9.807,148.910
C06289=1143.485,382.995,-85.075,-176.162,9.811,148.910
C06290=1143.481,383.242,-85.112,-176.161,9.815,148.911
C06291=1143.478,383.490,-85.149,-176.160,9.818,148.912
C06292=1143.474,383.737,-85.186,-176.159,9.822,148.912
C06293=1143.470,383.984,-85.223,-176.158,9.825,148.913
C06294=1143.466,384.231,-85.261,-176.158,9.828,148.914
C06295=1143.463,384.478,-85.297,-176.157,9.831,148.914
C06296=1143.459,384.725,-85.334,-176.157,9.835,148.915
C06297=1143.455,384.973,-85.371,-176.156,9.838,148.916
C06298=1143.451,385.220,-85.408,-176.156,9.841,148.916
C06299=1143.447,385.468,-85.445,-176.155,9.844,148.917
C06300=1143.443,385.714,-85.483,-176.155,9.847,148.918
C06301=1143.439,385.961,-85.520,-176.154,9.850,148.918
C06302=1143.435,386.209,-85.556,-176.154,9.853,148.919
C06303=1143.433,386.456,-85.593,-176.154,9.856,148.920
C06304=1143.428,386.703,-85.630,-176.154,9.859,148.921
C06305=1143.425,386.950,-85.668,-176.154,9.863,148.922
C06306=1143.421,387.197,-85.704,-176.154,9.865,148.922
C06307=1143.417,387.445,-85.742,-176.154,9.868,148.923
C06308=1143.413,387.692,-85.778,-176.154,9.870,148.924
C06309=1143.409,387.939,-85.816,-176.154,9.873,148.924
C06310=1143.406,388.187,-85.853,-176.154,9.877,148.925
C06311=1143.402,388.434,-85.890,-176.154,9.879,148.926
C06312=1143.397,388.681,-85.927,-176.155,9.882,148.927
C06313=1143.394,388.927,-85.964,-176.155,9.885,148.928
C06314=1143.391,389.175,-86.001,-176.156,9.886,148.928
C06315=1143.387,389.422,-86.038,-176.156,9.889,148.929
C06316=1143.383,389.670,-86.075,-176.156,9.892,148.930
C06317=1143.380,389.917,-86.113,-176.157,9.895,148.931
C06318=1143.375,390.164,-86.150,-176.157,9.897,148.932
C06319=1143.371,390.411,-86.187,-176.158,9.899,148.932
C06320=1143.367,390.698,-86.231,-176.158,9.902,148.933
C06321=1143.363,390.985,-86.273,-176.159,9.905,148.934
C06322=1143.358,391.273,-86.316,-176.160,9.908,148.935
C06323=1143.354,391.559,-86.359,-176.160,9.911,148.936
C06324=1143.350,391.806,-86.396,-176.161,9.913,148.937
C06325=1143.346,392.054,-86.433,-176.162,9.916,148.938
C06326=1143.343,392.301,-86.471,-176.163,9.918,148.939
C06327=1143.339,392.548,-86.508,-176.163,9.921,148.939
C06328=1143.335,392.796,-86.545,-176.164,9.923,148.940
C06329=1143.331,393.043,-86.583,-176.165,9.925,148.941
C06330=1143.327,393.290,-86.620,-176.166,9.928,148.942
C06331=1143.324,393.538,-86.657,-176.167,9.930,148.943
C06332=1143.320,393.784,-86.694,-176.168,9.932,148.943
C06333=1143.316,394.031,-86.731,-176.169,9.934,148.944
C06334=1143.312,394.279,-86.768,-176.170,9.936,148.945
C06335=1143.309,394.526,-86.806,-176.170,9.938,148.946
C06336=1143.305,394.773,-86.842,-176.171,9.940,148.947
C06337=1143.301,395.020,-86.879,-176.172,9.942,148.947
C06338=1143.298,395.267,-86.917,-176.174,9.945,148.948
C06339=1143.294,395.514,-86.954,-176.175,9.947,148.949
C06340=1143.290,395.762,-86.991,-176.176,9.949,148.950
C06341=1143.286,396.009,-87.028,-176.177,9.951,148.951
C06342=1143.282,396.256,-87.066,-176.178,9.953,148.952
C06343=1143.278,396.503,-87.102,-176.179,9.955,148.952
C06344=1143.274,396.750,-87.139,-176.180,9.957,148.953
C06345=1143.271,396.998,-87.177,-176.181,9.959,148.954
C06346=1143.267,397.245,-87.214,-176.182,9.961,148.955
C06347=1143.263,397.492,-87.251,-176.183,9.963,148.956
C06348=1143.260,397.739,-87.289,-176.184,9.965,148.957
C06349=1143.256,397.986,-87.326,-176.186,9.967,148.957
C06350=1143.252,398.234,-87.363,-176.187,9.970,148.959
C06351=1143.248,398.481,-87.401,-176.188,9.972,148.959
C06352=1143.244,398.728,-87.437,-176.189,9.974,148.960
C06353=1143.240,398.975,-87.474,-176.190,9.976,148.961
C06354=1143.236,399.222,-87.512,-176.191,9.978,148.962
C06355=1143.233,399.470,-87.549,-176.193,9.980,148.963
C06356=1143.229,399.717,-87.586,-176.194,9.981,148.963
C06357=1143.225,399.964,-87.623,-176.195,9.983,148.964
C06358=1143.221,400.211,-87.661,-176.196,9.985,148.965
C06359=1143.217,400.459,-87.698,-176.198,9.987,148.966
C06360=1143.214,400.705,-87.735,-176.199,9.989,148.967
C06361=1143.210,400.953,-87.772,-176.200,9.991,148.968
C06362=1143.206,401.200,-87.809,-176.201,9.994,148.968
C06363=1143.202,401.447,-87.846,-176.202,9.995,148.969
C06364=1143.198,401.694,-87.884,-176.204,9.997,148.970
C06365=1143.195,401.942,-87.921,-176.205,9.999,148.971
C06366=1143.191,402.189,-87.957,-176.206,10.001,148.972
C06367=1143.187,402.435,-87.995,-176.207,10.003,148.973
C06368=1143.184,402.683,-88.032,-176.208,10.005,148.973
C06369=1143.180,402.930,-88.069,-176.210,10.006,148.974
C06370=1143.176,403.177,-88.106,-176.211,10.008,148.975
C06371=1143.173,403.425,-88.144,-176.212,10.010,148.976
C06372=1143.169,403.672,-88.180,-176.213,10.013,148.977
C06373=1143.165,403.919,-88.218,-176.214,10.015,148.978
C06374=1143.161,404.166,-88.255,-176.215,10.017,148.978
C06375=1143.157,404.414,-88.292,-176.216,10.019,148.979
C06376=1143.153,404.660,-88.330,-176.218,10.020,148.980
C06377=1143.149,404.908,-88.367,-176.219,10.022,148.981
C06378=1143.146,405.155,-88.404,-176.220,10.024,148.982
C06379=1143.142,405.402,-88.441,-176.221,10.026,148.982
C06380=1143.138,405.649,-88.478,-176.222,10.028,148.983
C06381=1143.134,405.897,-88.515,-176.223,10.030,148.984
C06382=1143.131,406.144,-88.553,-176.224,10.032,148.985
C06383=1143.127,406.391,-88.590,-176.225,10.034,148.986
C06384=1143.122,406.638,-88.627,-176.227,10.036,148.987
C06385=1143.119,406.886,-88.664,-176.228,10.037,148.987
C06386=1143.115,407.132,-88.701,-176.229,10.040,148.988
C06387=1143.111,407.380,-88.738,-176.230,10.042,148.989
C06388=1143.108,407.628,-88.776,-176.231,10.044,148.990
C06389=1143.104,407.874,-88.813,-176.232,10.046,148.991
C06390=1143.100,408.121,-88.850,-176.233,10.048,148.991
C06391=1143.096,408.369,-88.887,-176.234,10.050,148.992
C06392=1143.092,408.616,-88.925,-176.235,10.052,148.993
C06393=1143.089,408.863,-88.961,-176.236,10.054,148.994
C06394=1143.085,409.110,-88.998,-176.237,10.056,148.994
C06395=1143.082,409.357,-89.036,-176.238,10.058,148.995
C06396=1143.078,409.604,-89.073,-176.239,10.060,148.996
C06397=1143.074,409.852,-89.110,-176.240,10.062,148.997
C06398=1143.070,410.099,-89.148,-176.241,10.064,148.998
C06399=1143.066,410.346,-89.184,-176.242,10.066,148.998
C06400=1143.062,410.593,-89.221,-176.243,10.068,148.999
C06401=1143.059,410.840,-89.259,-176.244,10.070,149.000
C06402=1143.055,411.088,-89.296,-176.245,10.072,149.001
C06403=1143.051,411.335,-89.333,-176.246,10.074,149.002
C06404=1143.047,411.581,-89.370,-176.247,10.076,149.002
C06405=1143.044,411.829,-89.408,-176.247,10.078,149.003
C06406=1143.039,412.076,-89.445,-176.248,10.080,149.004
C06407=1143.036,412.323,-89.482,-176.249,10.082,149.005
C06408=1143.032,412.571,-89.519,-176.250,10.084,149.005
C06409=1143.028,412.818,-89.556,-176.251,10.086,149.006
C06410=1143.024,413.065,-89.594,-176.252,10.088,149.007
C06411=1143.020,413.312,-89.631,-176.253,10.090,149.008
C06412=1143.017,413.560,-89.668,-176.253,10.093,149.009
C06413=1143.013,413.806,-89.705,-176.254,10.095,149.009
C06414=1143.009,414.054,-89.742,-176.255,10.097,149.010
C06415=1143.005,414.301,-89.780,-176.256,10.099,149.011
C06416=1143.002,414.548,-89.817,-176.257,10.101,149.011
C06417=1142.999,414.796,-89.854,-176.257,10.103,149.012
C06418=1142.996,415.043,-89.891,-176.258,10.105,149.013
C06419=1142.994,415.290,-89.928,-176.259,10.107,149.014
C06420=1142.992,415.537,-89.965,-176.260,10.109,149.014
C06421=1142.992,415.785,-90.001,-176.261,10.111,149.015
C06422=1142.993,416.032,-90.039,-176.261,10.114,149.016
C06423=1142.993,416.278,-90.075,-176.261,10.115,149.017
C06424=1142.995,416.533,-90.112,-176.263,10.117,149.017
C06425=1142.997,416.787,-90.150,-176.263,10.119,149.018
C06426=1143.001,417.040,-90.188,-176.264,10.121,149.019
C06427=1143.005,417.294,-90.224,-176.264,10.124,149.020
C06428=1142.584,417.296,-90.275,-176.266,10.134,149.023
C06429=1142.580,417.039,-90.238,-176.266,10.132,149.022
C06430=1142.577,416.782,-90.200,-176.265,10.131,149.022
C06431=1142.575,416.524,-90.161,-176.264,10.129,149.021
C06432=1142.573,416.267,-90.124,-176.264,10.126,149.020
C06433=1142.572,416.020,-90.087,-176.263,10.124,149.019
C06434=1142.572,415.773,-90.050,-176.262,10.122,149.019
C06435=1142.572,415.525,-90.013,-176.261,10.120,149.018
C06436=1142.573,415.279,-89.977,-176.261,10.118,149.017
C06437=1142.575,415.031,-89.939,-176.260,10.116,149.016
C06438=1142.578,414.784,-89.902,-176.259,10.114,149.016
C06439=1142.581,414.537,-89.865,-176.258,10.112,149.015
C06440=1142.585,414.289,-89.828,-176.258,10.110,149.014
C06441=1142.588,414.043,-89.791,-176.257,10.107,149.013
C06442=1142.592,413.795,-89.754,-176.256,10.105,149.012
C06443=1142.596,413.548,-89.716,-176.255,10.103,149.012
C06444=1142.600,413.301,-89.679,-176.254,10.101,149.011
C06445=1142.604,413.054,-89.642,-176.254,10.100,149.010
C06446=1142.607,412.806,-89.605,-176.253,10.097,149.010
C06447=1142.611,412.559,-89.567,-176.252,10.095,149.009
C06448=1142.615,412.312,-89.530,-176.251,10.092,149.008
C06449=1142.618,412.065,-89.492,-176.250,10.091,149.007
C06450=1142.622,411.818,-89.456,-176.249,10.089,149.006
C06451=1142.627,411.570,-89.419,-176.248,10.087,149.006
C06452=1142.630,411.323,-89.381,-176.248,10.085,149.005
C06453=1142.634,411.076,-89.344,-176.246,10.083,149.004
C06454=1142.638,410.829,-89.307,-176.245,10.081,149.003
C06455=1142.642,410.582,-89.269,-176.244,10.079,149.002
C06456=1142.645,410.334,-89.232,-176.244,10.077,149.002
C06457=1142.649,410.087,-89.195,-176.243,10.075,149.001
C06458=1142.653,409.841,-89.158,-176.242,10.072,149.000
C06459=1142.657,409.593,-89.121,-176.241,10.070,148.999
C06460=1142.661,409.345,-89.084,-176.240,10.068,148.998
C06461=1142.665,409.099,-89.046,-176.239,10.066,148.998
C06462=1142.668,408.851,-89.009,-176.238,10.064,148.997
C06463=1142.672,408.604,-88.972,-176.237,10.062,148.996
C06464=1142.676,408.357,-88.934,-176.235,10.061,148.995
C06465=1142.680,408.110,-88.898,-176.234,10.059,148.994
C06466=1142.683,407.862,-88.860,-176.233,10.057,148.994
C06467=1142.687,407.616,-88.823,-176.232,10.055,148.993
C06468=1142.691,407.368,-88.786,-176.231,10.052,148.992
C06469=1142.695,407.121,-88.749,-176.230,10.051,148.991
C06470=1142.699,406.874,-88.711,-176.229,10.049,148.991
C06471=1142.703,406.627,-88.674,-176.228,10.047,148.990
C06472=1142.706,406.379,-88.637,-176.227,10.045,148.989
C06473=1142.710,406.132,-88.600,-176.226,10.042,148.988
C06474=1142.714,405.885,-88.563,-176.225,10.040,148.987
C06475=1142.718,405.637,-88.525,-176.224,10.038,148.986
C06476=1142.721,405.391,-88.488,-176.223,10.036,148.986
C06477=1142.725,405.144,-88.452,-176.221,10.035,148.985
C06478=1142.729,404.897,-88.415,-176.220,10.033,148.984
C06479=1142.732,404.649,-88.377,-176.219,10.031,148.983
C06480=1142.736,404.402,-88.340,-176.218,10.029,148.982
C06481=1142.740,404.155,-88.303,-176.217,10.027,148.981
C06482=1142.743,403.908,-88.265,-176.216,10.025,148.981
C06483=1142.747,403.660,-88.228,-176.215,10.023,148.980
C06484=1142.752,403.413,-88.191,-176.213,10.021,148.979
C06485=1142.755,403.166,-88.153,-176.212,10.019,148.978
C06486=1142.759,402.919,-88.117,-176.211,10.017,148.977
C06487=1142.763,402.672,-88.080,-176.210,10.015,148.977
C06488=1142.766,402.424,-88.042,-176.209,10.013,148.976
C06489=1142.770,402.177,-88.005,-176.207,10.011,148.975
C06490=1142.774,401.930,-87.968,-176.206,10.010,148.974
C06491=1142.778,401.683,-87.931,-176.205,10.008,148.973
C06492=1142.782,401.436,-87.893,-176.204,10.006,148.972
C06493=1142.786,401.188,-87.856,-176.203,10.004,148.972
C06494=1142.789,400.942,-87.819,-176.201,10.002,148.971
C06495=1142.793,400.694,-87.782,-176.200,9.999,148.970
C06496=1142.797,400.447,-87.745,-176.199,9.997,148.969
C06497=1142.801,400.200,-87.707,-176.197,9.996,148.968
C06498=1142.804,399.952,-87.670,-176.196,9.994,148.967
C06499=1142.808,399.705,-87.633,-176.195,9.992,148.966
C06500=1142.812,399.458,-87.596,-176.194,9.990,148.966
C06501=1142.816,399.211,-87.559,-176.193,9.988,148.965
C06502=1142.820,398.963,-87.521,-176.192,9.986,148.964
C06503=1142.824,398.717,-87.484,-176.191,9.983,148.963
C06504=1142.828,398.470,-87.447,-176.190,9.981,148.962
C06505=1142.831,398.222,-87.410,-176.188,9.980,148.961
C06506=1142.835,397.975,-87.372,-176.187,9.978,148.961
C06507=1142.839,397.728,-87.335,-176.186,9.976,148.960
C06508=1142.843,397.480,-87.298,-176.185,9.974,148.959
C06509=1142.846,397.234,-87.261,-176.183,9.972,148.958
C06510=1142.850,396.986,-87.224,-176.182,9.970,148.957
C06511=1142.854,396.738,-87.187,-176.181,9.968,148.956
C06512=1142.858,396.492,-87.149,-176.180,9.966,148.956
C06513=1142.862,396.245,-87.112,-176.179,9.964,148.955
C06514=1142.866,395.997,-87.075,-176.178,9.962,148.954
C06515=1142.868,395.751,-87.038,-176.177,9.960,148.953
C06516=1142.872,395.503,-87.001,-176.176,9.957,148.952
C06517=1142.877,395.256,-86.964,-176.175,9.955,148.951
C06518=1142.880,395.009,-86.926,-176.174,9.953,148.951
C06519=1142.884,394.762,-86.889,-176.173,9.950,148.950
C06520=1142.888,394.514,-86.853,-176.172,9.948,148.949
C06521=1142.891,394.267,-86.815,-176.171,9.946,148.948
C06522=1142.895,394.020,-86.778,-176.170,9.944,148.947
C06523=1142.899,393.773,-86.741,-176.169,9.942,148.946
C06524=1142.903,393.526,-86.703,-176.168,9.939,148.946
C06525=1142.907,393.278,-86.666,-176.167,9.937,148.945
C06526=1142.911,393.031,-86.629,-176.166,9.936,148.944
C06527=1142.914,392.785,-86.592,-176.166,9.933,148.943
C06528=1142.918,392.537,-86.554,-176.165,9.931,148.942
C06529=1142.922,392.290,-86.518,-176.164,9.929,148.942
C06530=1142.926,392.042,-86.481,-176.163,9.926,148.941
C06531=1142.929,391.795,-86.443,-176.163,9.924,148.940
C06532=1142.933,391.548,-86.406,-176.162,9.921,148.939
C06533=1142.938,391.261,-86.364,-176.161,9.919,148.938
C06534=1142.942,390.974,-86.319,-176.160,9.916,148.937
C06535=1142.947,390.687,-86.277,-176.160,9.913,148.936
C06536=1142.951,390.400,-86.233,-176.159,9.910,148.935
C06537=1142.955,390.153,-86.196,-176.159,9.907,148.934
C06538=1142.958,389.905,-86.159,-176.158,9.905,148.934
C06539=1142.962,389.658,-86.121,-176.157,9.903,148.933
C06540=1142.966,389.411,-86.085,-176.157,9.900,148.932
C06541=1142.970,389.163,-86.047,-176.157,9.897,148.931
C06542=1142.974,388.916,-86.010,-176.157,9.895,148.931
C06543=1142.978,388.669,-85.973,-176.156,9.892,148.930
C06544=1142.981,388.423,-85.937,-176.156,9.889,148.929
C06545=1142.984,388.175,-85.899,-176.156,9.887,148.928
C06546=1142.989,387.928,-85.863,-176.155,9.884,148.928
C06547=1142.992,387.681,-85.825,-176.155,9.881,148.927
C06548=1142.996,387.433,-85.788,-176.155,9.879,148.926
C06549=1143.000,387.186,-85.751,-176.155,9.876,148.925
C06550=1143.004,386.939,-85.713,-176.156,9.873,148.925
C06551=1143.008,386.692,-85.676,-176.156,9.870,148.924
C06552=1143.011,386.444,-85.639,-176.156,9.867,148.923
C06553=1143.015,386.197,-85.602,-176.156,9.864,148.923
C06554=1143.019,385.950,-85.566,-176.156,9.861,148.922
C06555=1143.022,385.703,-85.528,-176.156,9.858,148.921
C06556=1143.026,385.456,-85.491,-176.157,9.855,148.920
C06557=1143.030,385.208,-85.454,-176.157,9.851,148.920
C06558=1143.034,384.961,-85.418,-176.157,9.849,148.919
C06559=1143.038,384.713,-85.380,-176.158,9.846,148.918
C06560=1143.042,384.467,-85.343,-176.159,9.842,148.918
C06561=1143.046,384.220,-85.306,-176.159,9.839,148.917
C06562=1143.050,383.972,-85.269,-176.160,9.836,148.916
C06563=1143.052,383.725,-85.232,-176.161,9.833,148.915
C06564=1143.057,383.478,-85.196,-176.162,9.829,148.915
C06565=1143.061,383.231,-85.159,-176.163,9.825,148.914
C06566=1143.064,382.984,-85.121,-176.164,9.822,148.914
C06567=1143.068,382.736,-85.084,-176.165,9.818,148.913
C06568=1143.072,382.489,-85.047,-176.166,9.815,148.912
C06569=1143.076,382.242,-85.010,-176.167,9.811,148.912
C06570=1143.079,381.995,-84.974,-176.168,9.808,148.911
C06571=1143.084,381.748,-84.937,-176.169,9.804,148.910
C06572=1143.087,381.500,-84.900,-176.171,9.800,148.910
C06573=1143.091,381.253,-84.863,-176.172,9.796,148.909
C06574=1143.095,381.005,-84.826,-176.173,9.793,148.909
C06575=1143.099,380.758,-84.790,-176.175,9.790,148.908
C06576=1143.103,380.511,-84.753,-176.177,9.786,148.908
C06577=1143.106,380.263,-84.716,-176.178,9.782,148.907
C06578=1143.110,380.016,-84.679,-176.180,9.778,148.906
C06579=1143.114,379.769,-84.643,-176.181,9.774,148.906
C06580=1143.118,379.522,-84.606,-176.183,9.771,148.905
C06581=1143.122,379.275,-84.569,-176.185,9.766,148.905
C06582=1143.125,379.027,-84.532,-176.187,9.762,148.904
C06583=1143.129,378.780,-84.496,-176.189,9.759,148.904
C06584=1143.133,378.533,-84.459,-176.191,9.755,148.903
C06585=1143.137,378.286,-84.422,-176.193,9.750,148.903
C06586=1143.141,378.039,-84.385,-176.195,9.747,148.902
C06587=1143.144,377.792,-84.349,-176.196,9.743,148.902
C06588=1143.148,377.544,-84.312,-176.199,9.739,148.901
C06589=1143.152,377.296,-84.275,-176.201,9.735,148.901
C06590=1143.156,377.049,-84.239,-176.203,9.730,148.900
C06591=1143.160,376.802,-84.202,-176.205,9.727,148.900
C06592=1143.164,376.555,-84.165,-176.207,9.722,148.899
C06593=1143.167,376.308,-84.129,-176.209,9.719,148.899
C06594=1143.172,376.060,-84.093,-176.211,9.714,148.898
C06595=1143.176,375.813,-84.056,-176.214,9.710,148.898
C06596=1143.179,375.566,-84.020,-176.216,9.706,148.897
C06597=1143.183,375.319,-83.983,-176.218,9.702,148.897
C06598=1143.186,375.071,-83.947,-176.221,9.697,148.896
C06599=1143.190,374.823,-83.910,-176.222,9.694,148.896
C06600=1143.194,374.576,-83.873,-176.225,9.689,148.895
C06601=1143.198,374.329,-83.837,-176.228,9.685,148.895
C06602=1143.202,374.081,-83.801,-176.230,9.681,148.894
C06603=1143.205,373.835,-83.765,-176.232,9.677,148.894
C06604=1143.210,373.587,-83.728,-176.234,9.673,148.893
C06605=1143.213,373.340,-83.692,-176.237,9.668,148.893
C06606=1143.217,373.093,-83.655,-176.239,9.664,148.893
C06607=1143.221,372.845,-83.620,-176.242,9.659,148.892
C06608=1143.225,372.598,-83.583,-176.244,9.656,148.892
C06609=1143.229,372.351,-83.547,-176.247,9.652,148.891
C06610=1143.233,372.103,-83.511,-176.249,9.647,148.891
C06611=1143.236,371.856,-83.474,-176.252,9.643,148.890
C06612=1143.241,371.609,-83.438,-176.254,9.639,148.890
C06613=1143.244,371.362,-83.402,-176.257,9.635,148.890
C06614=1143.248,371.114,-83.366,-176.260,9.630,148.889
C06615=1143.252,370.867,-83.329,-176.262,9.626,148.889
C06616=1143.256,370.619,-83.293,-176.265,9.621,148.888
C06617=1143.260,370.372,-83.258,-176.267,9.618,148.888
C06618=1143.263,370.125,-83.222,-176.270,9.614,148.888
C06619=1143.267,369.877,-83.185,-176.272,9.609,148.887
C06620=1143.271,369.630,-83.149,-176.275,9.605,148.887
C06621=1143.275,369.382,-83.113,-176.278,9.601,148.886
C06622=1143.279,369.135,-83.077,-176.280,9.597,148.886
C06623=1143.282,368.888,-83.041,-176.283,9.592,148.886
C06624=1143.287,368.640,-83.005,-176.286,9.588,148.885
C06625=1143.290,368.393,-82.969,-176.288,9.584,148.885
C06626=1143.294,368.146,-82.933,-176.291,9.580,148.885
C06627=1143.298,367.898,-82.897,-176.293,9.575,148.884
C06628=1143.302,367.651,-82.862,-176.296,9.571,148.884
C06629=1143.305,367.403,-82.826,-176.299,9.567,148.883
C06630=1143.309,367.156,-82.789,-176.302,9.563,148.883
C06631=1143.314,366.909,-82.754,-176.304,9.558,148.883
C06632=1143.317,366.662,-82.718,-176.306,9.555,148.882
C06633=1143.322,366.414,-82.682,-176.309,9.551,148.882
C06634=1143.325,366.166,-82.647,-176.312,9.546,148.881
C06635=1143.329,365.919,-82.610,-176.315,9.542,148.881
C06636=1143.333,365.672,-82.575,-176.317,9.538,148.881
C06637=1143.338,365.388,-82.534,-176.320,9.533,148.880
C06638=1143.342,365.105,-82.493,-176.323,9.529,148.880
C06639=1143.346,364.821,-82.452,-176.326,9.523,148.879
C06640=1143.351,364.537,-82.412,-176.330,9.518,148.879
C06641=1143.355,364.290,-82.376,-176.332,9.515,148.879
C06642=1143.358,364.043,-82.340,-176.334,9.510,148.878
C06643=1143.363,363.795,-82.304,-176.337,9.506,148.878
C06644=1143.366,363.548,-82.268,-176.340,9.502,148.877
C06645=1143.370,363.300,-82.233,-176.342,9.498,148.877
C06646=1143.374,363.053,-82.197,-176.345,9.494,148.877
C06647=1143.378,362.805,-82.163,-176.348,9.489,148.877
C06648=1143.382,362.558,-82.127,-176.350,9.486,148.876
C06649=1143.386,362.310,-82.092,-176.353,9.482,148.876
C06650=1143.389,362.063,-82.056,-176.355,9.477,148.875
C06651=1143.394,361.815,-82.020,-176.358,9.473,148.875
C06652=1143.398,361.568,-81.985,-176.361,9.469,148.875
C06653=1143.402,361.321,-81.949,-176.363,9.465,148.874
C06654=1143.405,361.073,-81.914,-176.366,9.461,148.874
C06655=1143.409,360.826,-81.878,-176.368,9.457,148.874
C06656=1143.413,360.578,-81.843,-176.371,9.453,148.873
C06657=1143.417,360.331,-81.808,-176.373,9.448,148.873
C06658=1143.421,360.083,-81.773,-176.376,9.445,148.873
C06659=1143.424,359.836,-81.737,-176.378,9.441,148.872
C06660=1143.428,359.588,-81.702,-176.381,9.437,148.872
C06661=1143.433,359.341,-81.667,-176.384,9.432,148.871
C06662=1143.436,359.093,-81.632,-176.386,9.429,148.871
C06663=1143.440,358.846,-81.596,-176.389,9.425,148.871
C06664=1143.445,358.598,-81.562,-176.391,9.421,148.870
C06665=1143.448,358.351,-81.526,-176.394,9.416,148.870
C06666=1143.452,358.103,-81.490,-176.396,9.413,148.870
C06667=1143.456,357.855,-81.456,-176.399,9.409,148.869
C06668=1143.460,357.608,-81.420,-176.401,9.404,148.869
C06669=1143.464,357.361,-81.385,-176.404,9.401,148.869
C06670=1143.467,357.113,-81.351,-176.406,9.397,148.868
C06671=1143.471,356.866,-81.315,-176.409,9.392,148.868
C06672=1143.475,356.618,-81.281,-176.411,9.389,148.868
C06673=1143.479,356.371,-81.245,-176.414,9.385,148.867
C06674=1143.483,356.123,-81.211,-176.416,9.380,148.867
C06675=1143.487,355.876,-81.175,-176.419,9.376,148.867
C06676=1143.491,355.628,-81.140,-176.421,9.373,148.866
C06677=1143.495,355.381,-81.105,-176.424,9.369,148.866
C06678=1143.499,355.133,-81.071,-176.427,9.364,148.865
C06679=1143.503,354.886,-81.036,-176.429,9.361,148.865
C06680=1143.507,354.638,-81.001,-176.432,9.357,148.865
C06681=1143.510,354.391,-80.965,-176.434,9.352,148.864
C06682=1143.515,354.143,-80.931,-176.436,9.349,148.864
C06683=1143.519,353.896,-80.895,-176.439,9.345,148.864
C06684=1143.523,353.649,-80.861,-176.442,9.341,148.863
C06685=1143.527,353.401,-80.827,-176.444,9.337,148.863
C06686=1143.530,353.153,-80.791,-176.447,9.333,148.863
C06687=1143.535,352.906,-80.757,-176.449,9.328,148.862
C06688=1143.538,352.658,-80.722,-176.451,9.325,148.862
C06689=1143.542,352.411,-80.687,-176.454,9.321,148.862
C06690=1143.546,352.163,-80.652,-176.457,9.317,148.861
C06691=1143.551,351.915,-80.618,-176.459,9.313,148.861
C06692=1143.554,351.668,-80.583,-176.462,9.309,148.861
C06693=1143.558,351.420,-80.548,-176.465,9.305,148.860
C06694=1143.562,351.173,-80.514,-176.467,9.301,148.860
C06695=1143.566,350.925,-80.479,-176.469,9.297,148.860
C06696=1143.570,350.678,-80.444,-176.471,9.294,148.859
C06697=1143.574,350.430,-80.409,-176.474,9.290,148.859
C06698=1143.578,350.183,-80.375,-176.477,9.285,148.859
C06699=1143.581,349.935,-80.341,-176.479,9.282,148.858
C06700=1143.586,349.687,-80.306,-176.482,9.278,148.858
C06701=1143.590,349.439,-80.271,-176.485,9.274,148.858
C06702=1143.594,349.192,-80.237,-176.487,9.270,148.858
C06703=1143.598,348.945,-80.202,-176.489,9.266,148.857
C06704=1143.601,348.698,-80.168,-176.492,9.262,148.857
C06705=1143.605,348.449,-80.133,-176.494,9.258,148.856
C06706=1143.610,348.202,-80.099,-176.497,9.254,148.856
C06707=1143.613,347.954,-80.064,-176.499,9.251,148.856
C06708=1143.618,347.707,-80.030,-176.502,9.247,148.856
C06709=1143.622,347.460,-79.996,-176.505,9.242,148.855
C06710=1143.625,347.212,-79.961,-176.507,9.239,148.855
C06711=1143.630,346.964,-79.927,-176.510,9.235,148.855
C06712=1143.633,346.716,-79.893,-176.512,9.230,148.854
C06713=1143.638,346.469,-79.858,-176.515,9.227,148.854
C06714=1143.641,346.221,-79.824,-176.517,9.223,148.854
C06715=1143.646,345.974,-79.789,-176.519,9.219,148.853
C06716=1143.649,345.727,-79.756,-176.522,9.215,148.853
C06717=1143.654,345.478,-79.721,-176.525,9.211,148.853
C06718=1143.658,345.231,-79.688,-176.527,9.208,148.852
C06719=1143.662,344.983,-79.653,-176.530,9.204,148.852
C06720=1143.665,344.735,-79.619,-176.532,9.200,148.852
C06721=1143.670,344.488,-79.584,-176.535,9.196,148.852
C06722=1143.673,344.240,-79.550,-176.538,9.192,148.851
C06723=1143.678,343.993,-79.516,-176.540,9.188,148.851
C06724=1143.682,343.745,-79.483,-176.543,9.184,148.851
C06725=1143.685,343.497,-79.448,-176.545,9.181,148.850
C06726=1143.690,343.250,-79.414,-176.547,9.177,148.850
C06727=1143.693,343.002,-79.380,-176.550,9.173,148.850
C06728=1143.698,342.754,-79.346,-176.553,9.169,148.850
C06729=1143.702,342.507,-79.312,-176.555,9.165,148.849
C06730=1143.705,342.259,-79.278,-176.558,9.162,148.849
C06731=1143.710,342.011,-79.244,-176.560,9.158,148.849
C06732=1143.714,341.764,-79.210,-176.563,9.153,148.848
C06733=1143.718,341.516,-79.176,-176.565,9.150,148.848
C06734=1143.722,341.268,-79.142,-176.568,9.146,148.848
C06735=1143.726,341.021,-79.108,-176.570,9.142,148.847
C06736=1143.730,340.774,-79.074,-176.573,9.138,148.847
C06737=1143.734,340.525,-79.040,-176.576,9.134,148.847
C06738=1143.737,340.278,-79.006,-176.578,9.131,148.847
C06739=1143.742,340.030,-78.973,-176.581,9.126,148.846
C06740=1143.746,339.783,-78.939,-176.583,9.123,148.846
C06741=1143.751,339.502,-78.900,-176.586,9.119,148.846
C06742=1143.755,339.222,-78.862,-176.589,9.114,148.845
C06743=1143.760,338.941,-78.824,-176.592,9.110,148.845
C06744=1143.764,338.661,-78.785,-176.595,9.106,148.845
C06745=1143.769,338.413,-78.752,-176.597,9.102,148.844
C06746=1143.772,338.165,-78.718,-176.600,9.098,148.844
C06747=1143.776,337.917,-78.685,-176.603,9.094,148.844
C06748=1143.780,337.670,-78.650,-176.605,9.091,148.844
C06749=1143.785,337.422,-78.617,-176.608,9.086,148.843
C06750=1143.788,337.174,-78.584,-176.610,9.083,148.843
C06751=1143.792,336.927,-78.550,-176.613,9.079,148.843
C06752=1143.796,336.679,-78.517,-176.615,9.076,148.843
C06753=1143.800,336.432,-78.483,-176.618,9.071,148.842
C06754=1143.805,336.184,-78.449,-176.620,9.068,148.842
C06755=1143.808,335.935,-78.416,-176.623,9.064,148.842
C06756=1143.812,335.688,-78.382,-176.626,9.060,148.841
C06757=1143.816,335.441,-78.349,-176.628,9.057,148.841
C06758=1143.820,335.193,-78.315,-176.631,9.052,148.841
C06759=1143.825,334.945,-78.282,-176.633,9.049,148.841
C06760=1143.828,334.697,-78.248,-176.636,9.045,148.840
C06761=1143.832,334.450,-78.215,-176.638,9.042,148.840
C06762=1143.836,334.202,-78.182,-176.641,9.037,148.840
C06763=1143.841,333.954,-78.148,-176.643,9.034,148.840
C06764=1143.845,333.707,-78.114,-176.646,9.030,148.839
C06765=1143.849,333.459,-78.081,-176.648,9.027,148.839
C06766=1143.853,333.211,-78.048,-176.651,9.023,148.839
C06767=1143.857,332.963,-78.014,-176.654,9.019,148.839
C06768=1143.861,332.715,-77.981,-176.656,9.015,148.838
C06769=1143.865,332.467,-77.948,-176.658,9.012,148.838
C06770=1143.869,332.220,-77.915,-176.661,9.008,148.838
C06771=1143.873,331.972,-77.882,-176.664,9.004,148.838
C06772=1143.877,331.725,-77.848,-176.667,9.000,148.837
C06773=1143.881,331.477,-77.815,-176.669,8.997,148.837
C06774=1143.885,331.229,-77.781,-176.671,8.993,148.837
C06775=1143.889,330.982,-77.748,-176.674,8.988,148.837
C06776=1143.893,330.733,-77.715,-176.677,8.985,148.836
C06777=1143.897,330.485,-77.682,-176.679,8.981,148.836
C06778=1143.901,330.238,-77.649,-176.682,8.978,148.836
C06779=1143.905,329.990,-77.616,-176.685,8.974,148.836
C06780=1143.909,329.743,-77.583,-176.687,8.970,148.835
C06781=1143.913,329.495,-77.550,-176.690,8.966,148.835
C06782=1143.917,329.247,-77.517,-176.692,8.963,148.835
C06783=1143.922,328.999,-77.484,-176.695,8.959,148.835
C06784=1143.926,328.751,-77.451,-176.697,8.955,148.834
C06785=1143.930,328.503,-77.418,-176.700,8.951,148.834
C06786=1143.934,328.256,-77.384,-176.702,8.948,148.834
C06787=1143.938,328.008,-77.351,-176.705,8.945,148.834
C06788=1143.941,327.760,-77.319,-176.708,8.941,148.834
C06789=1143.946,327.513,-77.286,-176.710,8.938,148.833
C06790=1143.950,327.264,-77.253,-176.713,8.933,148.833
C06791=1143.954,327.017,-77.220,-176.715,8.930,148.833
C06792=1143.958,326.769,-77.187,-176.718,8.926,148.832
C06793=1143.962,326.522,-77.154,-176.720,8.923,148.832
C06794=1143.966,326.274,-77.121,-176.723,8.918,148.832
C06795=1143.970,326.025,-77.089,-176.725,8.915,148.832
C06796=1143.974,325.778,-77.056,-176.728,8.911,148.832
C06797=1143.979,325.530,-77.022,-176.731,8.908,148.831
C06798=1143.982,325.282,-76.991,-176.733,8.904,148.831
C06799=1143.986,325.034,-76.957,-176.736,8.901,148.831
C06800=1143.991,324.786,-76.924,-176.739,8.896,148.831
C06801=1143.995,324.538,-76.892,-176.741,8.893,148.831
C06802=1143.998,324.291,-76.859,-176.744,8.889,148.830
C06803=1144.003,324.043,-76.826,-176.746,8.886,148.830
C06804=1144.007,323.795,-76.794,-176.749,8.882,148.830
C06805=1144.011,323.548,-76.761,-176.752,8.878,148.830
C06806=1144.015,323.300,-76.729,-176.754,8.875,148.830
C06807=1144.020,323.052,-76.696,-176.757,8.871,148.829
C06808=1144.023,322.804,-76.663,-176.759,8.868,148.829
C06809=1144.027,322.556,-76.631,-176.762,8.864,148.829
C06810=1144.032,322.308,-76.598,-176.764,8.861,148.829
C06811=1144.035,322.060,-76.566,-176.767,8.856,148.828
C06812=1144.039,321.813,-76.533,-176.770,8.853,148.828
C06813=1144.043,321.565,-76.501,-176.773,8.849,148.828
C06814=1144.047,321.317,-76.468,-176.775,8.846,148.828
C06815=1144.052,321.069,-76.436,-176.778,8.842,148.828
C06816=1144.056,320.822,-76.403,-176.780,8.838,148.827
C06817=1144.060,320.573,-76.371,-176.783,8.835,148.827
C06818=1144.064,320.325,-76.339,-176.785,8.831,148.827
C06819=1144.068,320.078,-76.306,-176.788,8.828,148.827
C06820=1144.072,319.830,-76.274,-176.791,8.824,148.827
C06821=1144.076,319.581,-76.241,-176.793,8.821,148.826
C06822=1144.080,319.335,-76.209,-176.796,8.816,148.826
C06823=1144.085,319.086,-76.177,-176.798,8.813,148.826
C06824=1144.088,318.839,-76.144,-176.801,8.810,148.826
C06825=1144.092,318.590,-76.112,-176.804,8.806,148.826
C06826=1144.096,318.342,-76.080,-176.806,8.803,148.825
C06827=1144.101,318.095,-76.048,-176.809,8.799,148.825
C06828=1144.105,317.847,-76.015,-176.811,8.795,148.825
C06829=1144.109,317.599,-75.983,-176.814,8.791,148.825
C06830=1144.113,317.351,-75.951,-176.816,8.788,148.825
C06831=1144.117,317.103,-75.918,-176.819,8.785,148.824
C06832=1144.121,316.856,-75.886,-176.822,8.781,148.824
C06833=1144.126,316.607,-75.854,-176.824,8.778,148.824
C06834=1144.129,316.359,-75.822,-176.827,8.774,148.824
C06835=1144.133,316.111,-75.790,-176.830,8.770,148.824
C06836=1144.138,315.864,-75.758,-176.832,8.767,148.824
C06837=1144.142,315.616,-75.726,-176.835,8.763,148.823
C06838=1144.146,315.367,-75.694,-176.837,8.760,148.823
C06839=1144.150,315.120,-75.661,-176.840,8.756,148.823
C06840=1144.154,314.873,-75.630,-176.842,8.752,148.823
C06841=1144.158,314.624,-75.597,-176.845,8.749,148.823
C06842=1144.162,314.376,-75.565,-176.848,8.745,148.823
C06843=1144.166,314.128,-75.534,-176.850,8.742,148.822
C06844=1144.171,313.881,-75.502,-176.853,8.738,148.822
C06845=1144.175,313.603,-75.466,-176.856,8.735,148.822
C06846=1144.180,313.325,-75.430,-176.859,8.731,148.822
C06847=1144.185,313.048,-75.394,-176.862,8.727,148.822
C06848=1144.189,312.769,-75.359,-176.864,8.722,148.821
C06849=1144.194,312.521,-75.327,-176.868,8.719,148.821
C06850=1144.197,312.273,-75.295,-176.870,8.715,148.821
C06851=1144.202,312.026,-75.263,-176.872,8.712,148.821
C06852=1144.205,311.778,-75.232,-176.875,8.708,148.821
C06853=1144.210,311.529,-75.199,-176.878,8.705,148.821
C06854=1144.214,311.282,-75.168,-176.881,8.701,148.820
C06855=1144.218,311.034,-75.136,-176.883,8.698,148.820
C06856=1144.221,310.786,-75.104,-176.886,8.695,148.820
C06857=1144.227,310.538,-75.073,-176.889,8.690,148.820
C06858=1144.231,310.290,-75.041,-176.891,8.687,148.820
C06859=1144.235,310.042,-75.009,-176.893,8.684,148.820
C06860=1144.239,309.794,-74.977,-176.896,8.680,148.819
C06861=1144.242,309.546,-74.946,-176.899,8.677,148.819
C06862=1144.247,309.298,-74.915,-176.901,8.674,148.819
C06863=1144.251,309.050,-74.882,-176.904,8.670,148.819
C06864=1144.256,308.803,-74.851,-176.907,8.666,148.819
C06865=1144.259,308.555,-74.819,-176.910,8.663,148.819
C06866=1144.263,308.306,-74.788,-176.912,8.659,148.819
C06867=1144.268,308.059,-74.756,-176.915,8.656,148.818
C06868=1144.271,307.810,-74.725,-176.918,8.652,148.818
C06869=1144.276,307.563,-74.694,-176.920,8.649,148.818
C06870=1144.280,307.314,-74.661,-176.923,8.646,148.818
C06871=1144.285,307.067,-74.630,-176.926,8.642,148.818
C06872=1144.289,306.818,-74.599,-176.928,8.638,148.818
C06873=1144.293,306.571,-74.567,-176.930,8.635,148.817
C06874=1144.297,306.322,-74.536,-176.934,8.631,148.817
C06875=1144.301,306.074,-74.504,-176.936,8.628,148.817
C06876=1144.305,305.826,-74.474,-176.938,8.625,148.817
C06877=1144.309,305.578,-74.442,-176.941,8.621,148.817
C06878=1144.313,305.331,-74.410,-176.944,8.618,148.817
C06879=1144.317,305.082,-74.379,-176.946,8.615,148.817
C06880=1144.322,304.835,-74.348,-176.949,8.610,148.817
C06881=1144.326,304.586,-74.317,-176.952,8.607,148.816
C06882=1144.330,304.339,-74.285,-176.954,8.604,148.816
C06883=1144.334,304.090,-74.254,-176.957,8.600,148.816
C06884=1144.339,303.842,-74.223,-176.960,8.597,148.816
C06885=1144.343,303.595,-74.192,-176.962,8.594,148.816
C06886=1144.347,303.346,-74.161,-176.965,8.590,148.816
C06887=1144.351,303.099,-74.129,-176.968,8.587,148.816
C06888=1144.355,302.850,-74.098,-176.970,8.583,148.815
C06889=1144.360,302.602,-74.067,-176.973,8.580,148.815
C06890=1144.364,302.354,-74.035,-176.976,8.576,148.815
C06891=1144.368,302.106,-74.005,-176.978,8.573,148.815
C06892=1144.372,301.858,-73.973,-176.981,8.569,148.815
C06893=1144.377,301.610,-73.942,-176.984,8.566,148.815
C06894=1144.380,301.363,-73.912,-176.986,8.563,148.815
C06895=1144.384,301.114,-73.881,-176.989,8.560,148.815
C06896=1144.389,300.867,-73.849,-176.992,8.556,148.815
C06897=1144.393,300.618,-73.818,-176.994,8.553,148.814
C06898=1144.397,300.370,-73.787,-176.997,8.550,148.814
C06899=1144.402,300.122,-73.757,-177.000,8.546,148.814
C06900=1144.406,299.874,-73.725,-177.002,8.542,148.814
C06901=1144.410,299.626,-73.695,-177.005,8.539,148.814
C06902=1144.414,299.378,-73.663,-177.008,8.535,148.814
C06903=1144.418,299.130,-73.633,-177.010,8.532,148.814
C06904=1144.423,298.882,-73.602,-177.013,8.529,148.814
C06905=1144.426,298.634,-73.570,-177.015,8.526,148.814
C06906=1144.430,298.386,-73.540,-177.019,8.522,148.813
C06907=1144.435,298.138,-73.509,-177.021,8.519,148.813
C06908=1144.439,297.889,-73.478,-177.023,8.515,148.813
C06909=1144.444,297.642,-73.447,-177.027,8.512,148.813
C06910=1144.447,297.394,-73.417,-177.029,8.508,148.813
C06911=1144.451,297.145,-73.386,-177.031,8.505,148.813
C06912=1144.456,296.897,-73.355,-177.034,8.502,148.813
C06913=1144.461,296.649,-73.324,-177.037,8.498,148.813
C06914=1144.464,296.401,-73.294,-177.040,8.495,148.813
C06915=1144.469,296.153,-73.263,-177.042,8.492,148.812
C06916=1144.473,295.905,-73.232,-177.045,8.488,148.812
C06917=1144.476,295.657,-73.202,-177.048,8.485,148.812
C06918=1144.481,295.409,-73.171,-177.050,8.482,148.812
C06919=1144.486,295.161,-73.140,-177.053,8.479,148.812
C06920=1144.489,294.912,-73.110,-177.056,8.475,148.812
C06921=1144.494,294.664,-73.079,-177.058,8.471,148.812
C06922=1144.497,294.417,-73.049,-177.061,8.469,148.812
C06923=1144.502,294.169,-73.018,-177.063,8.465,148.812
C06924=1144.506,293.920,-72.987,-177.067,8.461,148.812
C06925=1144.510,293.673,-72.957,-177.069,8.458,148.811
C06926=1144.515,293.424,-72.927,-177.072,8.455,148.812
C06927=1144.519,293.176,-72.896,-177.074,8.452,148.811
C06928=1144.523,292.928,-72.865,-177.077,8.448,148.811
C06929=1144.527,292.680,-72.835,-177.080,8.445,148.811
C06930=1144.531,292.432,-72.804,-177.082,8.442,148.811
C06931=1144.536,292.183,-72.774,-177.085,8.439,148.811
C06932=1144.539,291.935,-72.744,-177.088,8.435,148.811
C06933=1144.544,291.687,-72.713,-177.090,8.432,148.811
C06934=1144.548,291.440,-72.683,-177.093,8.429,148.811
C06935=1144.553,291.191,-72.653,-177.096,8.426,148.811
C06936=1144.557,290.943,-72.623,-177.098,8.422,148.811
C06937=1144.561,290.695,-72.592,-177.101,8.419,148.811
C06938=1144.565,290.447,-72.561,-177.104,8.415,148.810
C06939=1144.570,290.198,-72.531,-177.106,8.412,148.810
C06940=1144.573,289.951,-72.501,-177.109,8.408,148.810
C06941=1144.577,289.703,-72.471,-177.112,8.405,148.810
C06942=1144.582,289.455,-72.441,-177.114,8.402,148.810
C06943=1144.586,289.206,-72.410,-177.117,8.399,148.810
C06944=1144.590,288.958,-72.380,-177.120,8.395,148.810
C06945=1144.594,288.710,-72.350,-177.123,8.392,148.810
C06946=1144.599,288.462,-72.319,-177.125,8.389,148.810
C06947=1144.603,288.214,-72.290,-177.128,8.386,148.810
C06948=1144.607,287.966,-72.260,-177.130,8.383,148.810
C06949=1144.612,287.690,-72.226,-177.134,8.379,148.810
C06950=1144.617,287.415,-72.193,-177.137,8.375,148.810
C06951=1144.621,287.139,-72.160,-177.140,8.371,148.810
C06952=1144.626,286.864,-72.126,-177.143,8.368,148.810
C06953=1144.630,286.616,-72.096,-177.145,8.365,148.809
C06954=1144.634,286.368,-72.066,-177.148,8.361,148.809
C06955=1144.639,286.119,-72.036,-177.151,8.358,148.809
C06956=1144.643,285.871,-72.006,-177.154,8.355,148.809
C06957=1144.647,285.623,-71.976,-177.156,8.352,148.809
C06958=1144.651,285.375,-71.946,-177.159,8.349,148.809
C06959=1144.656,285.126,-71.916,-177.162,8.345,148.809
C06960=1144.660,284.878,-71.887,-177.164,8.342,148.809
C06961=1144.664,284.631,-71.857,-177.167,8.338,148.809
C06962=1144.669,284.382,-71.827,-177.169,8.336,148.809
C06963=1144.673,284.134,-71.797,-177.172,8.333,148.809
C06964=1144.677,283.886,-71.767,-177.175,8.329,148.809
C06965=1144.681,283.638,-71.737,-177.178,8.326,148.809
C06966=1144.686,283.389,-71.707,-177.180,8.322,148.809
C06967=1144.690,283.142,-71.677,-177.183,8.319,148.809
C06968=1144.694,282.893,-71.648,-177.186,8.316,148.809
C06969=1144.698,282.645,-71.618,-177.189,8.312,148.808
C06970=1144.703,282.396,-71.588,-177.192,8.309,148.809
C06971=1144.707,282.148,-71.559,-177.194,8.306,148.808
C06972=1144.711,281.901,-71.529,-177.197,8.303,148.808
C06973=1144.715,281.652,-71.499,-177.199,8.300,148.808
C06974=1144.719,281.404,-71.470,-177.202,8.296,148.808
C06975=1144.724,281.156,-71.440,-177.205,8.293,148.808
C06976=1144.728,280.907,-71.410,-177.207,8.290,148.808
C06977=1144.733,280.659,-71.381,-177.210,8.287,148.808
C06978=1144.737,280.411,-71.351,-177.213,8.284,148.808
C06979=1144.741,280.163,-71.321,-177.215,8.281,148.808
C06980=1144.745,279.915,-71.292,-177.219,8.277,148.808
C06981=1144.749,279.666,-71.262,-177.221,8.274,148.808
C06982=1144.753,279.418,-71.233,-177.224,8.271,148.808
C06983=1144.757,279.170,-71.203,-177.227,8.268,148.808
C06984=1144.762,278.922,-71.174,-177.229,8.265,148.808
C06985=1144.766,278.674,-71.145,-177.232,8.262,148.808
C06986=1144.771,278.426,-71.115,-177.235,8.258,148.808
C06987=1144.775,278.178,-71.086,-177.237,8.255,148.808
C06988=1144.779,277.929,-71.056,-177.240,8.252,148.808
C06989=1144.783,277.681,-71.027,-177.243,8.249,148.808
C06990=1144.787,277.433,-70.998,-177.245,8.246,148.808
C06991=1144.791,277.184,-70.968,-177.248,8.243,148.808
C06992=1144.796,276.936,-70.939,-177.251,8.240,148.808
C06993=1144.800,276.688,-70.909,-177.254,8.236,148.808
C06994=1144.804,276.439,-70.880,-177.257,8.233,148.808
C06995=1144.809,276.191,-70.851,-177.259,8.230,148.808
C06996=1144.813,275.943,-70.822,-177.262,8.227,148.808
C06997=1144.817,275.695,-70.792,-177.264,8.224,148.808
C06998=1144.822,275.447,-70.763,-177.267,8.221,148.808
C06999=1144.826,275.198,-70.734,-177.270,8.217,148.808
C07000=1144.830,274.950,-70.704,-177.273,8.214,148.808
C07001=1144.835,274.701,-70.675,-177.276,8.211,148.808
C07002=1144.839,274.454,-70.646,-177.278,8.208,148.807
C07003=1144.843,274.205,-70.617,-177.281,8.205,148.807
C07004=1144.848,273.957,-70.587,-177.284,8.202,148.808
C07005=1144.852,273.708,-70.559,-177.286,8.198,148.807
C07006=1144.856,273.460,-70.530,-177.289,8.195,148.807
C07007=1144.860,273.213,-70.501,-177.292,8.192,148.807
C07008=1144.865,272.964,-70.472,-177.295,8.189,148.807
C07009=1144.869,272.716,-70.442,-177.297,8.186,148.807
C07010=1144.873,272.467,-70.413,-177.300,8.183,148.807
C07011=1144.878,272.218,-70.384,-177.303,8.180,148.807
C07012=1144.882,271.971,-70.356,-177.305,8.176,148.807
C07013=1144.886,271.723,-70.326,-177.308,8.173,148.807
C07014=1144.890,271.474,-70.298,-177.311,8.171,148.807
C07015=1144.895,271.226,-70.268,-177.313,8.168,148.807
C07016=1144.899,270.978,-70.239,-177.316,8.164,148.807
C07017=1144.903,270.730,-70.211,-177.319,8.161,148.807
C07018=1144.907,270.481,-70.181,-177.322,8.158,148.807
C07019=1144.912,270.232,-70.153,-177.325,8.155,148.807
C07020=1144.917,269.985,-70.124,-177.327,8.151,148.807
C07021=1144.920,269.736,-70.095,-177.330,8.149,148.807
C07022=1144.925,269.488,-70.066,-177.333,8.146,148.807
C07023=1144.929,269.239,-70.037,-177.335,8.143,148.807
C07024=1144.934,268.992,-70.008,-177.338,8.139,148.807
C07025=1144.938,268.743,-69.980,-177.341,8.136,148.807
C07026=1144.942,268.495,-69.951,-177.344,8.133,148.807
C07027=1144.947,268.247,-69.922,-177.347,8.130,148.807
C07028=1144.951,267.998,-69.894,-177.349,8.127,148.807
C07029=1144.955,267.750,-69.865,-177.352,8.124,148.807
C07030=1144.960,267.501,-69.836,-177.355,8.121,148.807
C07031=1144.963,267.254,-69.807,-177.357,8.118,148.807
C07032=1144.968,267.005,-69.779,-177.360,8.115,148.807
C07033=1144.973,266.756,-69.750,-177.362,8.112,148.807
C07034=1144.976,266.509,-69.721,-177.365,8.109,148.807
C07035=1144.981,266.260,-69.693,-177.368,8.106,148.807
C07036=1144.985,266.012,-69.665,-177.371,8.102,148.807
C07037=1144.989,265.763,-69.635,-177.374,8.099,148.807
C07038=1144.994,265.515,-69.607,-177.376,8.096,148.807
C07039=1144.998,265.267,-69.579,-177.379,8.093,148.807
C07040=1145.003,265.018,-69.550,-177.382,8.090,148.808
C07041=1145.007,264.771,-69.522,-177.385,8.087,148.808
C07042=1145.011,264.522,-69.493,-177.388,8.084,148.808
C07043=1145.015,264.273,-69.465,-177.390,8.081,148.807
C07044=1145.020,264.025,-69.436,-177.393,8.078,148.808
C07045=1145.024,263.776,-69.408,-177.396,8.075,148.808
C07046=1145.029,263.529,-69.379,-177.398,8.072,148.808
C07047=1145.033,263.280,-69.351,-177.401,8.069,148.808
C07048=1145.037,263.031,-69.322,-177.403,8.066,148.808
C07049=1145.042,262.783,-69.294,-177.406,8.063,148.808
C07050=1145.046,262.535,-69.266,-177.409,8.060,148.808
C07051=1145.051,262.286,-69.237,-177.412,8.056,148.808
C07052=1145.054,262.038,-69.209,-177.415,8.053,148.808
C07053=1145.059,261.765,-69.178,-177.418,8.050,148.808
C07054=1145.064,261.491,-69.147,-177.421,8.047,148.808
C07055=1145.069,261.218,-69.116,-177.424,8.044,148.808
C07056=1145.073,260.944,-69.085,-177.426,8.040,148.808
C07057=1145.078,260.696,-69.057,-177.429,8.038,148.808
C07058=1145.082,260.447,-69.028,-177.433,8.034,148.808
C07059=1145.087,260.199,-69.000,-177.435,8.031,148.808
C07060=1145.091,259.951,-68.972,-177.438,8.028,148.808
C07061=1145.095,259.703,-68.944,-177.441,8.025,148.808
C07062=1145.099,259.454,-68.915,-177.444,8.022,148.808
C07063=1145.104,259.206,-68.888,-177.446,8.019,148.808
C07064=1145.108,258.957,-68.859,-177.449,8.016,148.808
C07065=1145.113,258.709,-68.831,-177.452,8.013,148.808
C07066=1145.116,258.461,-68.803,-177.454,8.010,148.808
C07067=1145.121,258.212,-68.775,-177.457,8.007,148.808
C07068=1145.126,257.963,-68.747,-177.460,8.004,148.808
C07069=1145.130,257.715,-68.719,-177.463,8.001,148.808
C07070=1145.134,257.467,-68.692,-177.466,7.998,148.808
C07071=1145.139,257.219,-68.663,-177.468,7.995,148.808
C07072=1145.143,256.971,-68.635,-177.471,7.992,148.808
C07073=1145.147,256.722,-68.607,-177.473,7.989,148.808
C07074=1145.152,256.473,-68.579,-177.476,7.986,148.808
C07075=1145.156,256.225,-68.551,-177.479,7.983,148.809
C07076=1145.160,255.977,-68.523,-177.482,7.980,148.809
C07077=1145.164,255.728,-68.495,-177.485,7.977,148.809
C07078=1145.169,255.479,-68.468,-177.487,7.975,148.809
C07079=1145.174,255.232,-68.440,-177.490,7.972,148.809
C07080=1145.178,254.983,-68.412,-177.493,7.969,148.809
C07081=1145.182,254.734,-68.385,-177.496,7.966,148.809
C07082=1145.186,254.486,-68.356,-177.499,7.963,148.809
C07083=1145.191,254.238,-68.328,-177.501,7.960,148.809
C07084=1145.196,253.989,-68.301,-177.504,7.957,148.809
C07085=1145.199,253.741,-68.273,-177.506,7.954,148.809
C07086=1145.204,253.493,-68.245,-177.509,7.951,148.809
C07087=1145.208,253.244,-68.218,-177.512,7.948,148.809
C07088=1145.212,252.996,-68.190,-177.515,7.945,148.809
C07089=1145.217,252.747,-68.163,-177.518,7.942,148.809
C07090=1145.222,252.499,-68.134,-177.520,7.939,148.809
C07091=1145.226,252.250,-68.106,-177.523,7.936,148.809
C07092=1145.230,252.002,-68.079,-177.526,7.933,148.809
C07093=1145.235,251.754,-68.051,-177.529,7.930,148.810
C07094=1145.239,251.505,-68.024,-177.532,7.927,148.810
C07095=1145.243,251.257,-67.996,-177.534,7.924,148.810
C07096=1145.248,251.009,-67.969,-177.537,7.922,148.810
C07097=1145.252,250.760,-67.941,-177.540,7.919,148.810
C07098=1145.256,250.511,-67.914,-177.543,7.916,148.810
C07099=1145.261,250.263,-67.887,-177.545,7.913,148.810
C07100=1145.265,250.014,-67.859,-177.548,7.910,148.810
C07101=1145.269,249.766,-67.832,-177.551,7.907,148.810
C07102=1145.274,249.518,-67.804,-177.554,7.904,148.810
C07103=1145.278,249.269,-67.777,-177.556,7.901,148.810
C07104=1145.282,249.020,-67.749,-177.559,7.898,148.810
C07105=1145.287,248.772,-67.722,-177.562,7.895,148.810
C07106=1145.291,248.524,-67.695,-177.565,7.892,148.810
C07107=1145.295,248.275,-67.667,-177.567,7.889,148.810
C07108=1145.300,248.027,-67.639,-177.570,7.886,148.810
C07109=1145.304,247.778,-67.612,-177.573,7.883,148.810
C07110=1145.309,247.530,-67.585,-177.576,7.880,148.811
C07111=1145.313,247.281,-67.557,-177.578,7.877,148.811
C07112=1145.317,247.033,-67.530,-177.581,7.874,148.811
C07113=1145.322,246.784,-67.503,-177.584,7.871,148.811
C07114=1145.327,246.536,-67.476,-177.586,7.869,148.811
C07115=1145.331,246.288,-67.448,-177.589,7.866,148.811
C07116=1145.335,246.039,-67.421,-177.592,7.864,148.811
C07117=1145.340,245.790,-67.394,-177.595,7.861,148.811
C07118=1145.344,245.542,-67.367,-177.597,7.858,148.811
C07119=1145.348,245.294,-67.340,-177.600,7.855,148.811
C07120=1145.353,245.046,-67.312,-177.603,7.852,148.811
C07121=1145.357,244.796,-67.285,-177.606,7.849,148.811
C07122=1145.361,244.548,-67.258,-177.609,7.846,148.811
C07123=1145.366,244.299,-67.231,-177.611,7.843,148.812
C07124=1145.370,244.051,-67.204,-177.615,7.840,148.812
C07125=1145.375,243.803,-67.177,-177.617,7.838,148.812
C07126=1145.379,243.554,-67.150,-177.620,7.835,148.812
C07127=1145.383,243.305,-67.123,-177.623,7.832,148.812
C07128=1145.388,243.057,-67.096,-177.626,7.829,148.812
C07129=1145.392,242.808,-67.069,-177.629,7.826,148.812
C07130=1145.397,242.560,-67.042,-177.631,7.823,148.812
C07131=1145.401,242.311,-67.015,-177.634,7.821,148.812
C07132=1145.406,242.063,-66.988,-177.636,7.818,148.812
C07133=1145.410,241.815,-66.962,-177.639,7.815,148.813
C07134=1145.415,241.566,-66.935,-177.642,7.812,148.813
C07135=1145.419,241.317,-66.907,-177.645,7.809,148.813
C07136=1145.423,241.069,-66.880,-177.648,7.806,148.813
C07137=1145.427,240.820,-66.854,-177.650,7.803,148.813
C07138=1145.432,240.572,-66.827,-177.653,7.800,148.813
C07139=1145.436,240.323,-66.800,-177.656,7.797,148.813
C07140=1145.440,240.075,-66.773,-177.659,7.795,148.813
C07141=1145.445,239.827,-66.746,-177.661,7.792,148.813
C07142=1145.450,239.578,-66.719,-177.664,7.789,148.813
C07143=1145.454,239.330,-66.692,-177.666,7.787,148.813
C07144=1145.459,239.081,-66.666,-177.670,7.784,148.814
C07145=1145.463,238.832,-66.639,-177.673,7.781,148.814
C07146=1145.467,238.584,-66.613,-177.675,7.778,148.814
C07147=1145.472,238.336,-66.586,-177.678,7.775,148.814
C07148=1145.476,238.087,-66.558,-177.681,7.772,148.814
C07149=1145.481,237.838,-66.533,-177.684,7.769,148.814
C07150=1145.485,237.590,-66.506,-177.686,7.766,148.814
C07151=1145.489,237.342,-66.479,-177.689,7.764,148.814
C07152=1145.494,237.093,-66.452,-177.691,7.761,148.814
C07153=1145.499,236.844,-66.426,-177.694,7.759,148.814
C07154=1145.503,236.596,-66.399,-177.697,7.756,148.814
C07155=1145.507,236.347,-66.372,-177.700,7.753,148.815
C07156=1145.512,236.099,-66.347,-177.703,7.750,148.815
C07157=1145.516,235.826,-66.317,-177.706,7.747,148.815
C07158=1145.521,235.555,-66.287,-177.709,7.743,148.815
C07159=1145.526,235.283,-66.259,-177.712,7.741,148.815
C07160=1145.531,235.011,-66.230,-177.715,7.738,148.815
C07161=1145.535,234.763,-66.204,-177.718,7.735,148.815
C07162=1145.540,234.514,-66.177,-177.721,7.732,148.816
C07163=1145.544,234.266,-66.151,-177.724,7.729,148.816
C07164=1145.549,234.017,-66.124,-177.726,7.727,148.816
C07165=1145.553,233.768,-66.098,-177.729,7.724,148.816
C07166=1145.558,233.519,-66.072,-177.731,7.721,148.816
C07167=1145.562,233.271,-66.045,-177.734,7.718,148.816
C07168=1145.567,233.022,-66.019,-177.737,7.715,148.816
C07169=1145.571,232.774,-65.992,-177.740,7.713,148.816
C07170=1145.575,232.525,-65.967,-177.743,7.710,148.816
C07171=1145.579,232.277,-65.940,-177.746,7.707,148.817
C07172=1145.584,232.028,-65.914,-177.748,7.705,148.817
C07173=1145.589,231.780,-65.887,-177.751,7.702,148.817
C07174=1145.593,231.531,-65.861,-177.754,7.699,148.817
C07175=1145.597,231.283,-65.835,-177.757,7.696,148.817
C07176=1145.602,231.034,-65.809,-177.760,7.694,148.817
C07177=1145.606,230.785,-65.783,-177.763,7.691,148.817
C07178=1145.611,230.537,-65.756,-177.765,7.689,148.817
C07179=1145.615,230.288,-65.730,-177.768,7.686,148.817
C07180=1145.620,230.040,-65.704,-177.770,7.683,148.818
C07181=1145.625,229.791,-65.678,-177.773,7.680,148.818
C07182=1145.629,229.542,-65.652,-177.776,7.677,148.818
C07183=1145.633,229.294,-65.625,-177.779,7.674,148.818
C07184=1145.637,229.045,-65.600,-177.781,7.672,148.818
C07185=1145.642,228.796,-65.573,-177.784,7.669,148.818
C07186=1145.646,228.547,-65.547,-177.787,7.666,148.818
C07187=1145.651,228.300,-65.521,-177.790,7.663,148.818
C07188=1145.656,228.051,-65.495,-177.793,7.661,148.819
C07189=1145.660,227.802,-65.469,-177.796,7.658,148.819
C07190=1145.664,227.553,-65.444,-177.798,7.656,148.819
C07191=1145.668,227.305,-65.417,-177.801,7.653,148.819
C07192=1145.673,227.057,-65.392,-177.804,7.650,148.819
C07193=1145.678,226.808,-65.365,-177.806,7.647,148.819
C07194=1145.682,226.559,-65.340,-177.810,7.644,148.819
C07195=1145.686,226.310,-65.314,-177.812,7.642,148.820
C07196=1145.691,226.062,-65.288,-177.815,7.639,148.820
C07197=1145.695,225.814,-65.262,-177.817,7.637,148.820
C07198=1145.700,225.565,-65.236,-177.820,7.634,148.820
C07199=1145.704,225.316,-65.210,-177.824,7.631,148.820
C07200=1145.708,225.067,-65.184,-177.826,7.628,148.820
C07201=1145.713,224.819,-65.159,-177.829,7.626,148.820
C07202=1145.718,224.570,-65.133,-177.831,7.623,148.820
C07203=1145.722,224.322,-65.107,-177.835,7.621,148.821
C07204=1145.727,224.073,-65.081,-177.837,7.618,148.821
C07205=1145.732,223.824,-65.056,-177.840,7.616,148.821
C07206=1145.736,223.575,-65.030,-177.842,7.613,148.821
C07207=1145.740,223.327,-65.004,-177.845,7.610,148.821
C07208=1145.745,223.079,-64.979,-177.848,7.607,148.821
C07209=1145.749,222.830,-64.953,-177.851,7.604,148.822
C07210=1145.753,222.581,-64.927,-177.853,7.602,148.822
C07211=1145.758,222.333,-64.902,-177.856,7.599,148.822
C07212=1145.762,222.084,-64.876,-177.860,7.597,148.822
C07213=1145.767,221.835,-64.850,-177.862,7.594,148.822
C07214=1145.771,221.587,-64.825,-177.865,7.591,148.822
C07215=1145.776,221.338,-64.799,-177.867,7.589,148.822
C07216=1145.780,221.089,-64.774,-177.870,7.586,148.822
C07217=1145.785,220.841,-64.749,-177.873,7.583,148.823
C07218=1145.789,220.592,-64.723,-177.876,7.580,148.823
C07219=1145.793,220.343,-64.697,-177.878,7.578,148.823
C07220=1145.798,220.095,-64.672,-177.881,7.575,148.823
C07221=1145.802,219.846,-64.646,-177.884,7.573,148.823
C07222=1145.807,219.597,-64.621,-177.887,7.570,148.824
C07223=1145.812,219.349,-64.596,-177.889,7.568,148.824
C07224=1145.816,219.100,-64.570,-177.893,7.565,148.824
C07225=1145.820,218.851,-64.544,-177.896,7.562,148.824
C07226=1145.825,218.603,-64.519,-177.898,7.559,148.824
C07227=1145.830,218.354,-64.494,-177.901,7.557,148.824
C07228=1145.834,218.106,-64.468,-177.904,7.555,148.825
C07229=1145.839,217.857,-64.443,-177.907,7.552,148.825
C07230=1145.843,217.607,-64.418,-177.909,7.549,148.825
C07231=1145.848,217.359,-64.392,-177.912,7.547,148.825
C07232=1145.852,217.110,-64.366,-177.915,7.544,148.825
C07233=1145.857,216.862,-64.342,-177.918,7.541,148.825
C07234=1145.861,216.613,-64.317,-177.920,7.538,148.825
C07235=1145.866,216.365,-64.291,-177.923,7.537,148.826
C07236=1145.870,216.116,-64.266,-177.926,7.534,148.826
C07237=1145.874,215.867,-64.240,-177.929,7.531,148.826
C07238=1145.879,215.619,-64.215,-177.932,7.528,148.826
C07239=1145.883,215.370,-64.191,-177.934,7.526,148.826
C07240=1145.888,215.122,-64.165,-177.937,7.523,148.826
C07241=1145.892,214.872,-64.140,-177.940,7.520,148.827
C07242=1145.897,214.624,-64.115,-177.942,7.518,148.827
C07243=1145.902,214.375,-64.090,-177.945,7.516,148.827
C07244=1145.906,214.127,-64.065,-177.948,7.513,148.827
C07245=1145.910,213.877,-64.040,-177.951,7.510,148.827
C07246=1145.915,213.629,-64.015,-177.954,7.508,148.828
C07247=1145.920,213.380,-63.989,-177.956,7.505,148.828
C07248=1145.924,213.132,-63.965,-177.960,7.502,148.828
C07249=1145.928,212.883,-63.940,-177.962,7.500,148.828
C07250=1145.933,212.635,-63.914,-177.965,7.497,148.828
C07251=1145.938,212.385,-63.889,-177.968,7.495,148.828
C07252=1145.942,212.137,-63.864,-177.970,7.493,148.829
C07253=1145.946,211.888,-63.839,-177.973,7.490,148.829
C07254=1145.951,211.639,-63.815,-177.976,7.487,148.829
C07255=1145.955,211.391,-63.790,-177.979,7.484,148.829
C07256=1145.960,211.142,-63.765,-177.981,7.482,148.829
C07257=1145.965,210.892,-63.740,-177.984,7.480,148.830
C07258=1145.969,210.644,-63.714,-177.987,7.477,148.830
C07259=1145.974,210.396,-63.690,-177.989,7.475,148.830
C07260=1145.978,210.147,-63.665,-177.993,7.472,148.830
C07261=1145.984,209.876,-63.639,-177.996,7.469,148.830
C07262=1145.988,209.606,-63.612,-177.999,7.467,148.831
C07263=1145.993,209.335,-63.585,-178.002,7.464,148.831
C07264=1145.998,209.064,-63.558,-178.005,7.461,148.831
C07265=1146.003,208.816,-63.532,-178.008,7.458,148.831
C07266=1146.007,208.567,-63.507,-178.010,7.456,148.831
C07267=1146.012,208.319,-63.483,-178.013,7.454,148.831
C07268=1146.016,208.069,-63.458,-178.016,7.451,148.832
C07269=1146.020,207.821,-63.434,-178.018,7.449,148.832
C07270=1146.025,207.573,-63.409,-178.021,7.446,148.832
C07271=1146.029,207.323,-63.384,-178.024,7.443,148.832
C07272=1146.034,207.075,-63.360,-178.027,7.441,148.832
C07273=1146.039,206.826,-63.336,-178.030,7.438,148.833
C07274=1146.043,206.577,-63.311,-178.033,7.436,148.833
C07275=1146.048,206.328,-63.286,-178.035,7.434,148.833
C07276=1146.053,206.080,-63.262,-178.038,7.431,148.833
C07277=1146.057,205.830,-63.237,-178.041,7.428,148.833
C07278=1146.061,205.583,-63.212,-178.044,7.426,148.834
C07279=1146.066,205.334,-63.187,-178.046,7.423,148.834
C07280=1146.070,205.085,-63.163,-178.050,7.421,148.834
C07281=1146.075,204.836,-63.138,-178.052,7.419,148.834
C07282=1146.080,204.588,-63.114,-178.055,7.416,148.834
C07283=1146.084,204.338,-63.090,-178.057,7.414,148.835
C07284=1146.089,204.090,-63.065,-178.060,7.411,148.835
C07285=1146.093,203.841,-63.041,-178.063,7.409,148.835
C07286=1146.098,203.592,-63.016,-178.066,7.406,148.835
C07287=1146.102,203.344,-62.992,-178.069,7.404,148.835
C07288=1146.107,203.095,-62.967,-178.072,7.401,148.836
C07289=1146.111,202.846,-62.943,-178.074,7.399,148.836
C07290=1146.116,202.597,-62.919,-178.077,7.396,148.836
C07291=1146.121,202.348,-62.895,-178.080,7.393,148.836
C07292=1146.125,202.099,-62.871,-178.083,7.392,148.836
C07293=1146.130,201.851,-62.847,-178.085,7.389,148.837
C07294=1146.134,201.602,-62.822,-178.088,7.387,148.837
C07295=1146.138,201.353,-62.797,-178.091,7.384,148.837
C07296=1146.143,201.105,-62.773,-178.094,7.382,148.837
C07297=1146.148,200.856,-62.749,-178.096,7.379,148.838
C07298=1146.152,200.606,-62.725,-178.099,7.377,148.838
C07299=1146.156,200.358,-62.701,-178.102,7.375,148.838
C07300=1146.162,200.109,-62.676,-178.105,7.372,148.838
C07301=1146.166,199.861,-62.652,-178.108,7.369,148.838
C07302=1146.170,199.612,-62.628,-178.110,7.367,148.839
C07303=1146.175,199.362,-62.604,-178.113,7.365,148.839
C07304=1146.180,199.114,-62.580,-178.116,7.363,148.839
C07305=1146.184,198.866,-62.556,-178.119,7.360,148.839
C07306=1146.188,198.617,-62.532,-178.122,7.357,148.839
C07307=1146.193,198.367,-62.507,-178.124,7.355,148.840
C07308=1146.198,198.119,-62.483,-178.127,7.352,148.840
C07309=1146.202,197.870,-62.459,-178.130,7.351,148.840
C07310=1146.207,197.621,-62.436,-178.133,7.348,148.840
C07311=1146.212,197.373,-62.411,-178.136,7.345,148.840
